Yaskawa INFORM job: DPRINT3D6.JBI

/JOB
//NAME DPRINT3D6
//POS
///NPOS 1000,0,0,0,0,0
///TOOL 9
///POSTYPE PULSE
///PULSE
C00000=29945,51705,-123586,60699,-119026,-94760,0
C00001=29937,51700,-123602,60705,-119017,-94763,0
C00002=29929,51696,-123618,60712,-119008,-94767,0
C00003=29921,51691,-123634,60719,-118999,-94770,0
C00004=29913,51687,-123649,60726,-118990,-94774,0
C00005=29905,51683,-123664,60732,-118981,-94777,0
C00006=29897,51678,-123679,60739,-118972,-94780,0
C00007=29889,51674,-123693,60746,-118964,-94782,0
C00008=29881,51670,-123708,60753,-118955,-94786,0
C00009=29873,51666,-123723,60760,-118947,-94789,0
C00010=29864,51662,-123736,60767,-118938,-94792,0
C00011=29856,51657,-123751,60774,-118930,-94795,0
C00012=29851,51655,-123762,60779,-118924,-94797,0
C00013=29843,51650,-123777,60786,-118915,-94800,0
C00014=29835,51646,-123793,60792,-118905,-94803,0
C00015=29827,51641,-123809,60799,-118896,-94807,0
C00016=29824,51639,-123816,60802,-118892,-94809,0
C00017=29807,51636,-123827,60819,-118882,-94809,0
C00018=29769,51629,-123849,60858,-118859,-94811,0
C00019=29726,51622,-123874,60903,-118835,-94812,0
C00020=29682,51615,-123900,60947,-118811,-94813,0
C00021=29646,51609,-123919,60985,-118791,-94814,0
C00022=29614,51604,-123934,61017,-118774,-94814,0
C00023=29583,51600,-123950,61050,-118758,-94814,0
C00024=29556,51596,-123961,61078,-118745,-94814,0
C00025=29529,51593,-123972,61107,-118731,-94814,0
C00026=29502,51590,-123982,61136,-118717,-94813,0
C00027=29474,51587,-123994,61164,-118704,-94813,0
C00028=29447,51583,-124005,61193,-118691,-94812,0
C00029=29424,51581,-124012,61218,-118680,-94812,0
C00030=29400,51579,-124020,61243,-118669,-94810,0
C00031=29377,51577,-124027,61267,-118658,-94810,0
C00032=29353,51574,-124035,61292,-118648,-94809,0
C00033=29333,51573,-124040,61314,-118639,-94807,0
C00034=29313,51571,-124046,61336,-118630,-94806,0
C00035=29292,51570,-124050,61358,-118622,-94805,0
C00036=29271,51568,-124055,61380,-118612,-94803,0
C00037=29251,51567,-124059,61402,-118603,-94802,0
C00038=29230,51565,-124065,61424,-118595,-94801,0
C00039=29210,51564,-124070,61446,-118586,-94800,0
C00040=29191,51563,-124073,61466,-118578,-94798,0
C00041=29173,51562,-124077,61486,-118571,-94797,0
C00042=29154,51560,-124081,61506,-118563,-94796,0
C00043=29132,51568,-124052,61533,-118568,-94785,0
C00044=29118,51573,-124034,61551,-118570,-94778,0
C00045=29103,51579,-124015,61570,-118573,-94770,0
C00046=29088,51585,-123994,61590,-118577,-94762,0
C00047=29072,51591,-123972,61610,-118580,-94754,0
C00048=29057,51597,-123951,61630,-118584,-94746,0
C00049=29042,51602,-123930,61649,-118587,-94738,0
C00050=29026,51608,-123909,61669,-118591,-94730,0
C00051=29011,51614,-123887,61689,-118594,-94722,0
C00052=28995,51621,-123864,61710,-118599,-94713,0
C00053=28978,51628,-123839,61731,-118603,-94704,0
C00054=28961,51635,-123812,61753,-118608,-94694,0
C00055=28944,51642,-123787,61775,-118612,-94684,0
C00056=28926,51650,-123758,61799,-118618,-94674,0
C00057=28907,51659,-123726,61824,-118625,-94662,0
C00058=28888,51668,-123694,61849,-118631,-94651,0
C00059=28869,51677,-123662,61874,-118638,-94639,0
C00060=28850,51686,-123631,61899,-118645,-94628,0
C00061=28831,51696,-123595,61925,-118651,-94615,0
C00062=28810,51707,-123556,61952,-118661,-94601,0
C00063=28789,51718,-123518,61980,-118669,-94588,0
C00064=28764,51733,-123464,62015,-118681,-94569,0
C00065=28738,51748,-123411,62050,-118694,-94550,0
C00066=28713,51763,-123358,62085,-118707,-94532,0
C00067=28711,51768,-123342,62089,-118712,-94527,0
C00068=28710,51773,-123323,62093,-118720,-94521,0
C00069=28708,51779,-123303,62097,-118727,-94516,0
C00070=28707,51784,-123284,62101,-118734,-94510,0
C00071=28705,51790,-123264,62105,-118742,-94504,0
C00072=28704,51796,-123245,62110,-118749,-94498,0
C00073=28703,51801,-123225,62114,-118756,-94492,0
C00074=28702,51807,-123204,62117,-118764,-94487,0
C00075=28701,51813,-123184,62121,-118772,-94481,0
C00076=28700,51819,-123163,62125,-118780,-94474,0
C00077=28699,51825,-123141,62128,-118788,-94468,0
C00078=28698,51831,-123121,62132,-118796,-94462,0
C00079=28697,51837,-123100,62136,-118804,-94456,0
C00080=28697,51843,-123078,62139,-118813,-94450,0
C00081=28696,51849,-123057,62143,-118822,-94444,0
C00082=28695,51855,-123035,62147,-118830,-94438,0
C00083=28694,51861,-123015,62150,-118838,-94431,0
C00084=28693,51867,-122994,62154,-118846,-94425,0
C00085=28693,51873,-122972,62158,-118854,-94419,0
C00086=28692,51880,-122949,62161,-118863,-94413,0
C00087=28692,51887,-122926,62164,-118872,-94406,0
C00088=28692,51893,-122903,62167,-118881,-94400,0
C00089=28692,51900,-122879,62170,-118890,-94393,0
C00090=28693,51907,-122854,62173,-118901,-94386,0
C00091=28694,51915,-122829,62176,-118911,-94379,0
C00092=28694,51922,-122805,62178,-118922,-94372,0
C00093=28695,51929,-122779,62181,-118931,-94364,0
C00094=28695,51936,-122754,62183,-118941,-94357,0
C00095=28696,51944,-122729,62186,-118951,-94350,0
C00096=28695,51949,-122708,62189,-118959,-94344,0
C00097=28697,51988,-122575,62205,-119012,-94307,0
C00098=28700,52060,-122326,62235,-119112,-94236,0
C00099=28703,52132,-122079,62265,-119211,-94166,0
C00100=22589,60303,-97251,72637,-124455,-86218,0
C00101=22532,60337,-97155,72711,-124447,-86182,0
C00102=22418,60406,-96963,72858,-124431,-86109,0
C00103=22305,60475,-96769,73005,-124414,-86036,0
C00104=22296,60482,-96752,73017,-124413,-86030,0
C00105=22287,60488,-96735,73029,-124412,-86024,0
C00106=22278,60494,-96718,73041,-124411,-86018,0
C00107=22269,60500,-96701,73053,-124411,-86011,0
C00108=22260,60506,-96684,73065,-124410,-86005,0
C00109=22251,60512,-96667,73077,-124409,-85998,0
C00110=22242,60519,-96650,73089,-124408,-85992,0
C00111=22233,60525,-96633,73101,-124408,-85986,0
C00112=22224,60531,-96615,73113,-124406,-85980,0
C00113=22215,60537,-96598,73125,-124405,-85973,0
C00114=22206,60543,-96581,73137,-124404,-85967,0
C00115=22197,60549,-96564,73149,-124404,-85961,0
C00116=22188,60555,-96547,73161,-124403,-85954,0
C00117=22180,60562,-96530,73172,-124402,-85949,0
C00118=22176,60564,-96522,73178,-124402,-85946,0
C00119=22166,60591,-96449,73200,-124414,-85924,0
C00120=22151,60635,-96326,73237,-124439,-85886,0
C00121=22136,60680,-96203,73274,-124462,-85849,0
C00122=22124,60716,-96103,73303,-124481,-85819,0
C00123=22117,60744,-96026,73324,-124496,-85795,0
C00124=22111,60768,-95959,73341,-124510,-85776,0
C00125=22106,60792,-95893,73358,-124525,-85756,0
C00126=22101,60816,-95827,73374,-124539,-85737,0
C00127=22096,60840,-95761,73391,-124552,-85717,0
C00128=22092,60858,-95711,73403,-124564,-85702,0
C00129=22090,60875,-95665,73414,-124574,-85689,0
C00130=22087,60891,-95622,73424,-124583,-85676,0
C00131=22086,60906,-95580,73433,-124594,-85665,0
C00132=22085,60921,-95539,73442,-124604,-85653,0
C00133=22083,60936,-95497,73450,-124613,-85641,0
C00134=22082,60951,-95457,73459,-124624,-85629,0
C00135=22082,60965,-95418,73466,-124634,-85618,0
C00136=22081,60979,-95379,73473,-124643,-85607,0
C00137=22081,60993,-95340,73481,-124653,-85596,0
C00138=22080,61008,-95301,73488,-124663,-85585,0
C00139=22080,61022,-95262,73496,-124673,-85574,0
C00140=22079,61036,-95223,73503,-124682,-85563,0
C00141=22079,61050,-95184,73511,-124693,-85552,0
C00142=22078,61064,-95145,73518,-124702,-85540,0
C00143=22078,61078,-95107,73525,-124712,-85530,0
C00144=22078,61092,-95070,73532,-124721,-85519,0
C00145=22077,61106,-95033,73539,-124730,-85509,0
C00146=22088,61115,-95008,73532,-124744,-85503,0
C00147=22099,61124,-94983,73526,-124757,-85498,0
C00148=22111,61133,-94958,73519,-124771,-85492,0
C00149=22123,61143,-94932,73512,-124785,-85487,0
C00150=22135,61152,-94906,73504,-124798,-85482,0
C00151=22147,61161,-94880,73497,-124813,-85477,0
C00152=22159,61171,-94854,73490,-124827,-85471,0
C00153=22171,61180,-94828,73483,-124841,-85466,0
C00154=22183,61190,-94802,73476,-124855,-85461,0
C00155=22195,61199,-94777,73468,-124870,-85455,0
C00156=22207,61209,-94751,73461,-124883,-85449,0
C00157=22219,61219,-94724,73453,-124898,-85444,0
C00158=22233,61228,-94698,73445,-124913,-85439,0
C00159=22246,61238,-94672,73436,-124928,-85434,0
C00160=22259,61248,-94645,73428,-124943,-85429,0
C00161=22277,61259,-94615,73416,-124961,-85423,0
C00162=22294,61270,-94584,73405,-124980,-85417,0
C00163=22311,61282,-94553,73393,-124999,-85411,0
C00164=22329,61293,-94522,73381,-125018,-85405,0
C00165=22346,61305,-94491,73370,-125036,-85399,0
C00166=22363,61316,-94460,73358,-125056,-85393,0
C00167=22382,61328,-94428,73345,-125075,-85387,0
C00168=22403,61340,-94395,73331,-125096,-85382,0
C00169=22428,61355,-94355,73312,-125122,-85375,0
C00170=22460,61371,-94309,73290,-125155,-85367,0
C00171=22491,61388,-94264,73267,-125186,-85359,0
C00172=22518,61402,-94226,73247,-125212,-85353,0
C00173=22552,61419,-94181,73222,-125244,-85346,0
C00174=22611,61443,-94117,73175,-125298,-85337,0
C00175=22617,61442,-94119,73169,-125300,-85339,0
C00176=22628,61441,-94122,73158,-125306,-85342,0
C00177=22639,61440,-94126,73146,-125312,-85344,0
C00178=22650,61438,-94129,73135,-125318,-85347,0
C00179=22661,61437,-94133,73123,-125325,-85350,0
C00180=22671,61436,-94136,73112,-125330,-85353,0
C00181=22682,61435,-94140,73100,-125336,-85356,0
C00182=22693,61433,-94143,73089,-125342,-85358,0
C00183=22704,61432,-94147,73077,-125348,-85361,0
C00184=22715,61431,-94150,73066,-125353,-85364,0
C00185=22726,61430,-94153,73054,-125359,-85367,0
C00186=22737,61429,-94157,73043,-125365,-85370,0
C00187=22854,61411,-94207,72918,-125423,-85404,0
C00188=22970,61393,-94257,72793,-125482,-85437,0
C00189=23087,61375,-94306,72668,-125542,-85470,0
C00190=38516,60450,-97093,77282,-121914,-85527,0
C00191=38540,60506,-96937,77284,-121963,-85486,0
C00192=38587,60619,-96625,77287,-122064,-85402,0
C00193=38635,60733,-96312,77291,-122166,-85319,0
C00194=38639,60742,-96286,77291,-122174,-85312,0
C00195=38643,60752,-96261,77291,-122183,-85306,0
C00196=38648,60761,-96236,77290,-122191,-85299,0
C00197=38652,60770,-96210,77290,-122200,-85292,0
C00198=38657,60779,-96185,77290,-122208,-85285,0
C00199=38661,60789,-96159,77290,-122217,-85279,0
C00200=38665,60798,-96134,77290,-122225,-85272,0
C00201=38670,60807,-96108,77289,-122235,-85266,0
C00202=38674,60816,-96083,77289,-122243,-85259,0
C00203=38679,60826,-96057,77289,-122251,-85252,0
C00204=38683,60835,-96032,77289,-122260,-85245,0
C00205=38687,60844,-96006,77289,-122268,-85238,0
C00206=38692,60854,-95981,77288,-122277,-85232,0
C00207=38696,60862,-95956,77288,-122285,-85226,0
C00208=38698,60867,-95944,77288,-122290,-85222,0
C00209=38725,60883,-95901,77269,-122316,-85213,0
C00210=38769,60909,-95831,77237,-122360,-85199,0
C00211=38814,60934,-95761,77204,-122403,-85186,0
C00212=38851,60954,-95706,77178,-122439,-85176,0
C00213=38879,60969,-95667,77156,-122466,-85168,0
C00214=38904,60981,-95636,77137,-122488,-85163,0
C00215=38929,60992,-95605,77118,-122510,-85158,0
C00216=38954,61003,-95574,77099,-122533,-85152,0
C00217=38978,61015,-95543,77080,-122555,-85147,0
C00218=38997,61023,-95521,77065,-122572,-85143,0
C00219=39015,61030,-95501,77051,-122587,-85140,0
C00220=39031,61037,-95483,77038,-122602,-85137,0
C00221=39047,61042,-95468,77025,-122616,-85135,0
C00222=39063,61048,-95453,77012,-122629,-85133,0
C00223=39079,61054,-95438,76999,-122642,-85131,0
C00224=39094,61059,-95424,76986,-122655,-85129,0
C00225=39110,61063,-95412,76974,-122668,-85128,0
C00226=39125,61068,-95399,76961,-122680,-85126,0
C00227=39140,61073,-95387,76948,-122692,-85125,0
C00228=39155,61077,-95375,76935,-122705,-85124,0
C00229=39170,61082,-95362,76923,-122717,-85122,0
C00230=39185,61087,-95349,76910,-122730,-85121,0
C00231=39200,61091,-95337,76897,-122741,-85119,0
C00232=39216,61096,-95325,76884,-122754,-85118,0
C00233=39230,61100,-95313,76872,-122767,-85117,0
C00234=39245,61104,-95302,76860,-122778,-85116,0
C00235=39259,61109,-95291,76847,-122790,-85115,0
C00236=39272,61102,-95309,76832,-122793,-85122,0
C00237=39285,61095,-95327,76816,-122796,-85129,0
C00238=39298,61088,-95347,76800,-122800,-85137,0
C00239=39312,61081,-95368,76783,-122805,-85144,0
C00240=39325,61074,-95388,76767,-122808,-85152,0
C00241=39339,61066,-95409,76750,-122811,-85161,0
C00242=39353,61059,-95429,76734,-122815,-85168,0
C00243=39366,61051,-95450,76717,-122818,-85176,0
C00244=39380,61044,-95470,76700,-122823,-85184,0
C00245=39393,61037,-95491,76684,-122826,-85192,0
C00246=39407,61029,-95511,76667,-122830,-85199,0
C00247=39421,61021,-95534,76650,-122833,-85208,0
C00248=39435,61013,-95557,76632,-122837,-85217,0
C00249=39449,61004,-95581,76614,-122840,-85226,0
C00250=39463,60996,-95604,76597,-122842,-85235,0
C00251=39481,60984,-95636,76575,-122846,-85246,0
C00252=39498,60973,-95668,76553,-122849,-85257,0
C00253=39515,60962,-95699,76531,-122853,-85269,0
C00254=39532,60950,-95731,76509,-122855,-85281,0
C00255=39549,60939,-95763,76487,-122859,-85292,0
C00256=39566,60927,-95794,76465,-122862,-85304,0
C00257=39584,60915,-95829,76441,-122864,-85317,0
C00258=39603,60901,-95868,76416,-122868,-85331,0
C00259=39626,60883,-95917,76386,-122870,-85348,0
C00260=39653,60861,-95978,76349,-122872,-85369,0
C00261=39680,60840,-96038,76313,-122875,-85391,0
C00262=39702,60821,-96089,76282,-122876,-85408,0
C00263=39730,60797,-96156,76244,-122877,-85432,0
C00264=39772,60754,-96276,76183,-122875,-85472,0
C00265=39773,60749,-96290,76180,-122872,-85476,0
C00266=39775,60739,-96316,76173,-122867,-85484,0
C00267=39777,60730,-96343,76167,-122862,-85492,0
C00268=39779,60720,-96369,76161,-122856,-85500,0
C00269=39781,60711,-96396,76155,-122852,-85508,0
C00270=39782,60701,-96422,76149,-122846,-85516,0
C00271=39784,60692,-96449,76143,-122841,-85524,0
C00272=39786,60682,-96475,76136,-122836,-85531,0
C00273=39788,60672,-96501,76130,-122831,-85539,0
C00274=39790,60663,-96528,76124,-122825,-85547,0
C00275=39792,60653,-96554,76118,-122821,-85555,0
C00276=39793,60644,-96581,76112,-122815,-85563,0
C00277=39808,60540,-96867,76051,-122755,-85647,0
C00278=39822,60438,-97152,75990,-122695,-85730,0
C00279=39836,60335,-97436,75930,-122636,-85814,0
C00280=30587,54971,-112893,83159,-114119,-89355,0
C00281=30599,54742,-113602,83076,-113987,-89576,0
C00282=26102,60146,-97730,68982,-126367,-86955,0
C00283=25840,59681,-99025,69012,-125831,-87267,0
C00284=25634,59454,-99658,69109,-125527,-87407,0
C00285=25332,58798,-101506,69089,-124805,-87871,0
C00286=25979,60253,-97431,69165,-126385,-86850,0
C00287=30587,54971,-112892,83159,-114119,-89355,0
C00288=31709,55377,-111663,82144,-114929,-89073,0
C00289=25839,57975,-103866,68149,-124352,-88615,0
C00290=26365,57183,-106175,67203,-123890,-89348,0
C00291=32807,55804,-110382,81171,-115756,-88784,0
C00292=33879,56254,-109050,80240,-116598,-88487,0
C00293=26912,56421,-108432,66247,-123417,-90067,0
C00294=27480,55689,-110642,65280,-122933,-90775,0
C00295=34926,56725,-107667,79351,-117457,-88183,0
C00296=35949,57218,-106233,78506,-118333,-87871,0
C00297=28070,54985,-112806,64301,-122438,-91471,0
C00298=28684,54309,-114927,63309,-121930,-92157,0
C00299=36947,57735,-104747,77703,-119224,-87551,0
C00300=37852,58236,-103319,76997,-120066,-87245,0
C00301=37910,58216,-103377,76930,-120084,-87270,0
C00302=29401,53804,-116547,62283,-121613,-92717,0
C00303=29691,53808,-116540,61968,-121730,-92760,0
C00304=30366,53748,-116745,61199,-121915,-92922,0
C00305=38739,58035,-103915,76018,-120418,-87536,0
C00306=38801,58025,-103945,75951,-120444,-87552,0
C00307=39443,58021,-103971,75297,-120792,-87646,0
C00308=39602,58044,-103908,75146,-120896,-87649,0
C00309=31268,53565,-117352,60117,-122023,-93230,0
C00310=31586,53466,-117679,59719,-122012,-93369,0
C00311=32325,53708,-116909,59020,-122601,-93280,0
C00312=40396,57540,-105383,74115,-120944,-88187,0
C00313=41188,56884,-107325,73008,-120835,-88860,0
C00314=33470,54107,-115653,57950,-123551,-93138,0
C00315=34587,54528,-114347,56920,-124521,-92992,0
C00316=42006,56254,-109216,71875,-120713,-89524,0
C00317=42851,55650,-111059,70716,-120580,-90176,0
C00318=35677,54970,-112991,55932,-125513,-92844,0
C00319=43402,51305,-125329,68233,-116168,-94477,0
C00320=43725,55072,-112853,69529,-120434,-90818,0
C00321=44627,54518,-114601,68312,-120275,-91449,0
C00322=44483,51740,-123805,67237,-117079,-94137,0
C00323=45527,52199,-122237,66296,-118013,-93796,0
C00324=45537,52695,-120546,66506,-118620,-93300,0
C00325=45537,52633,-120569,66515,-118645,-93280,0
C00326=46697,53753,-116919,65763,-120389,-92380,0
C00327=46484,53451,-117891,65855,-119960,-92629,0
C00328=46391,53159,-118843,65822,-119586,-92891,0
C00329=46413,52869,-119803,65666,-119250,-93171,0
C00330=46552,52597,-120719,65391,-118971,-93455,0
C00331=46800,52351,-121557,65008,-118755,-93730,0
C00332=31582,53062,-118822,59567,-121584,-93654,0
C00333=31079,53242,-118223,60209,-121640,-93412,0
C00334=30561,53361,-117825,60837,-121604,-93223,0
C00335=30009,53428,-117599,61476,-121481,-93076,0
C00336=29447,53437,-117559,62097,-121280,-92979,0
C00337=28896,53391,-117698,62679,-121012,-92936,0
C00338=24566,59142,-100391,70091,-124739,-87405,0
C00339=24937,59442,-99553,69860,-125191,-87233,0
C00340=25205,59777,-98620,69755,-125616,-87019,0
C00341=25384,60157,-97564,69765,-126028,-86756,0
C00342=25469,60567,-96432,69890,-126406,-86456,0
C00343=29650,54961,-112750,84133,-113691,-89204,0
C00344=37685,58554,-102273,77329,-120238,-86893,0
C00345=38136,58340,-102891,76787,-120350,-87132,0
C00346=38606,58212,-103267,76260,-120523,-87303,0
C00347=39106,58161,-103425,75733,-120765,-87417,0
C00348=39613,58188,-103358,75231,-121064,-87466,0
C00349=40132,58300,-103047,74754,-121431,-87448,0
C00350=46626,53790,-116798,65857,-120402,-92336,0
C00351=48080,52338,-121638,63597,-119184,-93923,0
C00352=31354,52451,-120852,59527,-120671,-94173,0
C00353=31201,52571,-120444,59753,-120784,-94039,0
C00354=30927,52714,-119961,60125,-120883,-93865,0
C00355=30607,52827,-119581,60531,-120921,-93713,0
C00356=30254,52906,-119311,60958,-120900,-93585,0
C00357=29878,52950,-119159,61393,-120821,-93487,0
C00358=29495,52956,-119132,61816,-120689,-93424,0
C00359=29122,52926,-119226,62211,-120513,-93395,0
C00360=29011,52905,-119293,62324,-120446,-93397,0
C00361=28935,52897,-119318,62403,-120407,-93394,0
C00362=28456,52795,-119645,62881,-120103,-93418,0
C00363=23544,59431,-99566,71281,-124398,-87003,0
C00364=23825,59520,-99321,71038,-124627,-86981,0
C00365=24097,59665,-98918,70832,-124897,-86913,0
C00366=24327,59854,-98395,70691,-125179,-86805,0
C00367=24510,60081,-97764,70620,-125464,-86660,0
C00368=24634,60340,-97049,70624,-125739,-86481,0
C00369=24696,60619,-96279,70704,-125995,-86277,0
C00370=24693,60909,-95482,70856,-126218,-86054,0
C00371=24624,61196,-94694,71073,-126396,-85821,0
C00372=28555,55200,-111997,85310,-113265,-88883,0
C00373=37805,59412,-99847,77570,-120870,-86202,0
C00374=37976,59213,-100409,77316,-120843,-86388,0
C00375=38214,59036,-100913,77004,-120864,-86567,0
C00376=38493,58902,-101297,76668,-120935,-86716,0
C00377=38807,58815,-101551,76316,-121054,-86832,0
C00378=39141,58780,-101658,75966,-121220,-86908,0
C00379=39481,58798,-101612,75632,-121426,-86942,0
C00380=39812,58871,-101412,75331,-121665,-86931,0
C00381=40119,58996,-101065,75077,-121928,-86874,0
C00382=40308,59117,-100727,74941,-122122,-86804,0
C00383=47910,53822,-116729,64476,-120945,-92502,0
C00384=47717,53706,-117098,64631,-120735,-92578,0
C00385=47517,53528,-117667,64766,-120449,-92711,0
C00386=47387,53338,-118283,64818,-120175,-92868,0
C00387=47331,53142,-118926,64789,-119919,-93044,0
C00388=47352,52947,-119570,64677,-119690,-93231,0
C00389=47450,52764,-120182,64485,-119502,-93420,0
C00390=47620,52599,-120739,64223,-119357,-93603,0
C00391=47693,52555,-120892,64122,-119327,-93657,0
C00392=47732,52522,-121003,64065,-119300,-93693,0
C00393=48011,52374,-121513,63690,-119207,-93878,0
C00394=48242,52920,-119683,63689,-119983,-93387,0
C00395=48338,52828,-119993,63541,-119902,-93488,0
C00396=48398,52792,-120115,63459,-119878,-93531,0
C00397=48426,52769,-120192,63417,-119859,-93557,0
C00398=48563,52696,-120443,63232,-119814,-93647,0
C00399=48728,52637,-120643,63024,-119797,-93727,0
C00400=48914,52596,-120787,62799,-119810,-93794,0
C00401=49115,52574,-120866,62568,-119851,-93844,0
C00402=49652,52569,-120900,61974,-120029,-93930,0
C00403=30732,51817,-123013,59918,-119564,-94680,0
C00404=30754,52010,-122343,59984,-119849,-94498,0
C00405=30718,52122,-121960,60075,-119995,-94386,0
C00406=30636,52229,-121591,60217,-120118,-94272,0
C00407=30516,52322,-121274,60393,-120205,-94167,0
C00408=30359,52403,-120996,60605,-120263,-94068,0
C00409=30175,52467,-120777,60838,-120286,-93980,0
C00410=29972,52511,-120623,61082,-120275,-93908,0
C00411=29757,52536,-120536,61330,-120233,-93853,0
C00412=29540,52539,-120521,61571,-120160,-93818,0
C00413=29329,52522,-120574,61795,-120064,-93802,0
C00414=29239,52506,-120627,61887,-120010,-93804,0
C00415=29184,52500,-120645,61944,-119983,-93802,0
C00416=28994,52461,-120775,62135,-119863,-93812,0
C00417=28822,52404,-120962,62298,-119728,-93840,0
C00418=28675,52334,-121198,62426,-119583,-93887,0
C00419=28559,52252,-121475,62516,-119434,-93949,0
C00420=28349,52018,-122269,62640,-119049,-94147,0
C00421=22462,60078,-97747,72692,-124270,-86314,0
C00422=22881,59971,-98051,72218,-124434,-86468,0
C00423=23049,59957,-98090,72041,-124521,-86506,0
C00424=23127,59964,-98072,71965,-124572,-86514,0
C00425=23172,59963,-98076,71919,-124597,-86522,0
C00426=23344,59987,-98011,71757,-124716,-86532,0
C00427=23510,60040,-97866,71615,-124852,-86519,0
C00428=23662,60123,-97638,71502,-125005,-86481,0
C00429=23793,60231,-97341,71423,-125164,-86419,0
C00430=23898,60361,-96980,71383,-125327,-86336,0
C00431=23971,60511,-96568,71384,-125484,-86232,0
C00432=24009,60673,-96122,71427,-125630,-86114,0
C00433=24009,60842,-95658,71512,-125759,-85984,0
C00434=23971,61010,-95195,71636,-125862,-85848,0
C00435=23919,61122,-94888,71746,-125915,-85752,0
C00436=23874,61195,-94688,71828,-125943,-85689,0
C00437=23749,61329,-94321,72021,-125966,-85564,0
C00438=23379,61600,-93579,72527,-125937,-85292,0
C00439=38290,60454,-96953,77539,-121827,-85431,0
C00440=38275,60082,-97984,77393,-121581,-85727,0
C00441=38302,59941,-98375,77305,-121507,-85843,0
C00442=38330,59880,-98546,77251,-121484,-85896,0
C00443=38339,59843,-98649,77226,-121467,-85928,0
C00444=38410,59712,-99017,77099,-121423,-86044,0
C00445=38513,59593,-99352,76946,-121407,-86155,0
C00446=38647,59493,-99635,76769,-121419,-86255,0
C00447=38804,59416,-99855,76579,-121460,-86340,0
C00448=38982,59366,-100000,76381,-121530,-86406,0
C00449=39172,59345,-100061,76182,-121627,-86450,0
C00450=39366,59356,-100035,75993,-121746,-86470,0
C00451=39557,59399,-99918,75821,-121886,-86463,0
C00452=39736,59473,-99714,75675,-122041,-86430,0
C00453=39847,59544,-99515,75597,-122155,-86389,0
C00454=39915,59600,-99361,75553,-122233,-86354,0
C00455=40028,59737,-98979,75503,-122394,-86261,0
C00456=40217,60115,-97929,75486,-122764,-85987,0
C00457=49320,53737,-117041,62893,-121389,-92800,0
C00458=48930,53677,-117223,63292,-121168,-92792,0
C00459=48720,53621,-117399,63495,-121020,-92810,0
C00460=48536,53546,-117638,63661,-120859,-92850,0
C00461=48384,53455,-117930,63784,-120692,-92910,0
C00462=48270,53353,-118260,63860,-120526,-92987,0
C00463=48199,53245,-118611,63888,-120367,-93077,0
C00464=48169,53132,-118979,63868,-120219,-93176,0
C00465=48184,53023,-119341,63801,-120090,-93281,0
C00466=48214,52969,-119521,63742,-120034,-93336,0
C00467=48109,52838,-119955,63796,-119832,-93446,0
C00468=49394,53547,-117657,62721,-121185,-92983,0
C00469=49490,53541,-117679,62612,-121214,-93003,0
C00470=49683,53530,-117722,62395,-121272,-93044,0
C00471=49785,53524,-117745,62280,-121303,-93066,0
C00472=49799,53522,-117748,62265,-121306,-93069,0
C00473=49813,53521,-117753,62249,-121309,-93072,0
C00474=49827,53520,-117756,62233,-121313,-93075,0
C00475=49840,53519,-117761,62217,-121318,-93079,0
C00476=49852,53518,-117764,62204,-121320,-93082,0
C00477=49863,53517,-117769,62191,-121322,-93085,0
C00478=49876,53515,-117774,62176,-121326,-93088,0
C00479=49889,53514,-117779,62161,-121329,-93091,0
C00480=49903,53512,-117784,62146,-121331,-93095,0
C00481=49916,53511,-117790,62130,-121335,-93098,0
C00482=49929,53509,-117794,62115,-121338,-93101,0
C00483=49943,53508,-117800,62099,-121342,-93105,0
C00484=49956,53506,-117805,62084,-121344,-93108,0
C00485=49969,53505,-117810,62069,-121347,-93112,0
C00486=49983,53503,-117815,62053,-121351,-93115,0
C00487=49993,53502,-117819,62042,-121353,-93118,0
C00488=50003,53501,-117824,62030,-121354,-93121,0
C00489=50045,53479,-117898,61973,-121343,-93148,0
C00490=50081,53458,-117964,61923,-121330,-93172,0
C00491=50118,53438,-118031,61873,-121319,-93196,0
C00492=50148,53421,-118090,61831,-121307,-93216,0
C00493=50173,53406,-118138,61797,-121298,-93234,0
C00494=50192,53393,-118181,61770,-121289,-93249,0
C00495=50212,53380,-118224,61742,-121280,-93264,0
C00496=50231,53367,-118268,61714,-121269,-93278,0
C00497=50251,53354,-118311,61686,-121260,-93294,0
C00498=50271,53341,-118354,61658,-121251,-93309,0
C00499=50283,53331,-118386,61639,-121243,-93319,0
C00500=50296,53322,-118417,61621,-121236,-93330,0
C00501=50309,53312,-118449,61602,-121228,-93341,0
C00502=50321,53303,-118480,61585,-121221,-93351,0
C00503=50332,53293,-118511,61568,-121213,-93361,0
C00504=50343,53284,-118541,61551,-121205,-93371,0
C00505=50355,53275,-118572,61534,-121197,-93382,0
C00506=50366,53265,-118603,61517,-121189,-93392,0
C00507=50377,53256,-118634,61500,-121181,-93402,0
C00508=50389,53247,-118665,61483,-121174,-93412,0
C00509=50399,53238,-118694,61467,-121166,-93422,0
C00510=50408,53229,-118723,61453,-121159,-93431,0
C00511=50417,53221,-118750,61439,-121151,-93440,0
C00512=50427,53213,-118778,61425,-121143,-93450,0
C00513=50436,53204,-118805,61411,-121136,-93458,0
C00514=50443,53197,-118831,61399,-121129,-93466,0
C00515=50450,53189,-118856,61387,-121121,-93475,0
C00516=50458,53182,-118881,61375,-121114,-93483,0
C00517=50465,53174,-118905,61364,-121107,-93491,0
C00518=50473,53166,-118931,61352,-121100,-93499,0
C00519=50480,53159,-118956,61340,-121093,-93507,0
C00520=50487,53151,-118981,61328,-121087,-93515,0
C00521=50495,53144,-119007,61317,-121078,-93523,0
C00522=50502,53136,-119031,61305,-121072,-93531,0
C00523=50497,53130,-119054,61307,-121061,-93537,0
C00524=50490,53120,-119084,61310,-121046,-93544,0
C00525=50483,53111,-119115,61314,-121033,-93551,0
C00526=50476,53102,-119144,61317,-121018,-93558,0
C00527=50469,53093,-119174,61321,-121003,-93566,0
C00528=50461,53084,-119204,61325,-120989,-93573,0
C00529=50451,53073,-119240,61330,-120970,-93581,0
C00530=50441,53062,-119277,61336,-120953,-93590,0
C00531=50431,53051,-119312,61342,-120935,-93598,0
C00532=50421,53040,-119348,61348,-120918,-93607,0
C00533=50412,53029,-119385,61353,-120899,-93616,0
C00534=50401,53018,-119420,61359,-120882,-93624,0
C00535=50390,53006,-119457,61366,-120862,-93632,0
C00536=50378,52995,-119496,61374,-120843,-93642,0
C00537=50366,52983,-119535,61382,-120823,-93650,0
C00538=50351,52970,-119579,61392,-120800,-93660,0
C00539=50335,52955,-119625,61403,-120776,-93671,0
C00540=50318,52941,-119672,61415,-120752,-93682,0
C00541=50301,52927,-119718,61427,-120728,-93692,0
C00542=50292,52924,-119729,61436,-120720,-93693,0
C00543=50282,52921,-119740,61444,-120712,-93695,0
C00544=50273,52917,-119750,61454,-120704,-93697,0
C00545=50263,52914,-119762,61463,-120697,-93698,0
C00546=50252,52911,-119772,61473,-120689,-93700,0
C00547=50241,52907,-119782,61483,-120680,-93701,0
C00548=50230,52904,-119794,61494,-120672,-93703,0
C00549=50220,52901,-119804,61504,-120664,-93704,0
C00550=50209,52897,-119816,61514,-120656,-93706,0
C00551=50198,52894,-119826,61525,-120648,-93707,0
C00552=50186,52891,-119836,61536,-120639,-93708,0
C00553=50175,52888,-119847,61548,-120631,-93709,0
C00554=50163,52884,-119857,61559,-120623,-93710,0
C00555=50152,52881,-119867,61570,-120614,-93711,0
C00556=50140,52878,-119878,61581,-120606,-93712,0
C00557=50128,52875,-119888,61592,-120598,-93714,0
C00558=50117,52872,-119897,61604,-120590,-93715,0
C00559=50105,52869,-119907,61615,-120582,-93716,0
C00560=50094,52865,-119918,61626,-120574,-93717,0
C00561=50082,52862,-119928,61638,-120565,-93718,0
C00562=50071,52859,-119939,61649,-120557,-93719,0
C00563=50059,52856,-119949,61660,-120549,-93721,0
C00564=50047,52853,-119959,61672,-120541,-93722,0
C00565=50034,52850,-119968,61684,-120533,-93723,0
C00566=50022,52847,-119978,61697,-120525,-93724,0
C00567=50008,52844,-119988,61710,-120515,-93725,0
C00568=49994,52841,-119998,61725,-120506,-93725,0
C00569=49979,52837,-120007,61740,-120497,-93726,0
C00570=49964,52834,-120018,61755,-120488,-93726,0
C00571=49949,52831,-120028,61770,-120479,-93727,0
C00572=49934,52828,-120037,61784,-120468,-93728,0
C00573=49919,52825,-120048,61799,-120459,-93728,0
C00574=49905,52822,-120058,61814,-120450,-93729,0
C00575=49890,52819,-120068,61829,-120441,-93730,0
C00576=49875,52816,-120078,61844,-120432,-93730,0
C00577=49858,52812,-120088,61861,-120421,-93730,0
C00578=49803,52804,-120115,61918,-120390,-93730,0
C00579=49709,52789,-120161,62014,-120340,-93730,0
C00580=30345,51835,-122941,60354,-119464,-94607,0
C00581=30254,51752,-123229,60417,-119316,-94675,0
C00582=30162,51670,-123514,60480,-119167,-94742,0
C00583=30155,51664,-123533,60486,-119156,-94747,0
C00584=30148,51658,-123553,60491,-119146,-94752,0
C00585=30141,51653,-123573,60496,-119135,-94756,0
C00586=30134,51647,-123593,60502,-119125,-94761,0
C00587=30127,51642,-123610,60507,-119116,-94765,0
C00588=30121,51637,-123626,60511,-119107,-94769,0
C00589=30114,51632,-123645,60517,-119097,-94773,0
C00590=30106,51627,-123663,60523,-119087,-94777,0
C00591=30098,51622,-123681,60529,-119077,-94781,0
C00592=30090,51616,-123701,60535,-119066,-94785,0
C00593=30083,51611,-123719,60541,-119056,-94789,0
C00594=30075,51605,-123739,60547,-119046,-94794,0
C00595=30067,51600,-123757,60553,-119035,-94798,0
C00596=30059,51594,-123776,60560,-119025,-94802,0
C00597=30051,51589,-123795,60566,-119015,-94807,0
C00598=30044,51584,-123811,60571,-119005,-94810,0
C00599=30038,51580,-123826,60576,-118997,-94814,0
C00600=30035,51578,-123833,60579,-118993,-94815,0
C00601=30003,51571,-123856,60611,-118973,-94817,0
C00602=29951,51561,-123890,60665,-118942,-94820,0
C00603=29898,51551,-123925,60718,-118910,-94823,0
C00604=29845,51541,-123959,60772,-118879,-94825,0
C00605=29807,51535,-123981,60811,-118857,-94827,0
C00606=29772,51529,-124000,60847,-118838,-94827,0
C00607=29739,51525,-124016,60882,-118820,-94827,0
C00608=29706,51520,-124032,60916,-118803,-94827,0
C00609=29674,51515,-124047,60950,-118787,-94827,0
C00610=29641,51511,-124063,60984,-118770,-94827,0
C00611=29613,51507,-124075,61013,-118755,-94827,0
C00612=29589,51505,-124084,61038,-118743,-94827,0
C00613=29566,51502,-124093,61063,-118732,-94826,0
C00614=29543,51499,-124101,61087,-118722,-94825,0
C00615=29520,51497,-124108,61111,-118711,-94824,0
C00616=29498,51495,-124115,61135,-118701,-94824,0
C00617=29475,51493,-124121,61159,-118691,-94823,0
C00618=29453,51491,-124128,61183,-118680,-94821,0
C00619=29430,51489,-124136,61206,-118670,-94821,0
C00620=29408,51487,-124142,61230,-118660,-94820,0
C00621=29385,51485,-124149,61254,-118650,-94818,0
C00622=29365,51484,-124154,61276,-118641,-94817,0
C00623=29345,51482,-124158,61297,-118633,-94816,0
C00624=29326,51481,-124163,61319,-118625,-94814,0
C00625=29306,51479,-124167,61340,-118616,-94813,0
C00626=29287,51478,-124171,61360,-118609,-94812,0
C00627=29269,51478,-124173,61379,-118602,-94810,0
C00628=29252,51477,-124177,61398,-118595,-94809,0
C00629=29234,51476,-124179,61417,-118588,-94807,0
C00630=29216,51475,-124181,61436,-118581,-94806,0
C00631=29199,51474,-124183,61456,-118574,-94804,0
C00632=29181,51473,-124186,61475,-118568,-94802,0
C00633=29164,51473,-124189,61494,-118561,-94800,0
C00634=29146,51472,-124192,61513,-118554,-94799,0
C00635=29137,51471,-124193,61522,-118550,-94798,0
C00636=29125,51475,-124178,61537,-118553,-94793,0
C00637=29110,51481,-124157,61556,-118556,-94785,0
C00638=29095,51487,-124135,61576,-118560,-94777,0
C00639=29080,51493,-124115,61595,-118563,-94769,0
C00640=29065,51499,-124093,61615,-118568,-94760,0
C00641=29050,51505,-124072,61634,-118571,-94752,0
C00642=29032,51513,-124044,61657,-118576,-94742,0
C00643=29015,51520,-124017,61680,-118581,-94733,0
C00644=28997,51528,-123989,61703,-118586,-94722,0
C00645=28980,51536,-123962,61725,-118592,-94712,0
C00646=28962,51543,-123935,61748,-118596,-94702,0
C00647=28945,51551,-123908,61771,-118602,-94692,0
C00648=28927,51559,-123878,61795,-118608,-94681,0
C00649=28908,51568,-123846,61819,-118615,-94670,0
C00650=28890,51577,-123813,61844,-118622,-94658,0
C00651=28870,51588,-123777,61870,-118630,-94645,0
C00652=28849,51599,-123736,61899,-118639,-94630,0
C00653=28827,51611,-123695,61928,-118648,-94616,0
C00654=28806,51622,-123654,61957,-118657,-94601,0
C00655=28803,51628,-123635,61962,-118664,-94596,0
C00656=28800,51633,-123618,61967,-118670,-94590,0
C00657=28798,51638,-123600,61973,-118677,-94585,0
C00658=28795,51643,-123581,61978,-118684,-94579,0
C00659=28793,51649,-123561,61983,-118691,-94574,0
C00660=28790,51654,-123541,61988,-118697,-94567,0
C00661=28788,51660,-123522,61993,-118704,-94561,0
C00662=28786,51666,-123502,61999,-118711,-94556,0
C00663=28783,51671,-123481,62004,-118719,-94550,0
C00664=28781,51677,-123462,62009,-118726,-94543,0
C00665=28780,51683,-123440,62013,-118734,-94537,0
C00666=28778,51689,-123419,62018,-118742,-94531,0
C00667=28776,51695,-123399,62023,-118749,-94525,0
C00668=28774,51701,-123378,62027,-118757,-94518,0
C00669=28772,51707,-123357,62032,-118765,-94513,0
C00670=28771,51713,-123335,62037,-118773,-94506,0
C00671=28769,51719,-123315,62041,-118780,-94500,0
C00672=28767,51725,-123294,62046,-118788,-94494,0
C00673=28765,51731,-123273,62051,-118796,-94488,0
C00674=28764,51737,-123253,62055,-118804,-94481,0
C00675=28762,51743,-123231,62060,-118811,-94475,0
C00676=28760,51749,-123210,62065,-118819,-94469,0
C00677=28759,51755,-123188,62069,-118827,-94463,0
C00678=28758,51761,-123166,62073,-118835,-94456,0
C00679=28756,51768,-123145,62077,-118845,-94450,0
C00680=28756,51774,-123122,62081,-118854,-94443,0
C00681=28755,51782,-123095,62085,-118863,-94435,0
C00682=28755,51789,-123070,62089,-118873,-94429,0
C00683=28754,51797,-123044,62093,-118884,-94421,0
C00684=28754,51804,-123018,62097,-118894,-94413,0
C00685=28753,51811,-122993,62101,-118904,-94406,0
C00686=28753,51819,-122967,62105,-118913,-94399,0
C00687=28752,51826,-122941,62108,-118924,-94391,0
C00688=28752,51834,-122915,62112,-118934,-94384,0
C00689=28752,51841,-122890,62116,-118944,-94376,0
C00690=28752,51849,-122861,62120,-118956,-94368,0
C00691=28756,51876,-122768,62128,-118994,-94343,0
C00692=28763,51921,-122611,62141,-119058,-94299,0
C00693=22641,60308,-97114,72623,-124545,-86164,0
C00694=22587,60350,-96995,72699,-124544,-86121,0
C00695=22478,60436,-96756,72849,-124543,-86037,0
C00696=22420,60483,-96627,72930,-124543,-85990,0
C00697=22412,60490,-96607,72942,-124543,-85984,0
C00698=22404,60497,-96587,72953,-124544,-85977,0
C00699=22396,60504,-96567,72965,-124544,-85970,0
C00700=22388,60511,-96548,72976,-124544,-85963,0
C00701=22380,60518,-96528,72988,-124545,-85956,0
C00702=22372,60526,-96508,73000,-124545,-85949,0
C00703=22364,60533,-96489,73011,-124545,-85942,0
C00704=22355,60540,-96469,73023,-124547,-85935,0
C00705=22347,60547,-96449,73034,-124547,-85929,0
C00706=22339,60554,-96429,73046,-124547,-85922,0
C00707=22333,60561,-96411,73055,-124548,-85915,0
C00708=22326,60567,-96393,73065,-124549,-85910,0
C00709=22319,60574,-96375,73075,-124549,-85903,0
C00710=22313,60580,-96357,73085,-124550,-85897,0
C00711=22306,60587,-96339,73094,-124551,-85891,0
C00712=22300,60593,-96320,73104,-124552,-85885,0
C00713=22294,60600,-96302,73113,-124554,-85878,0
C00714=22287,60607,-96282,73124,-124554,-85871,0
C00715=22279,60614,-96262,73135,-124555,-85865,0
C00716=22271,60622,-96242,73146,-124555,-85858,0
C00717=22264,60629,-96223,73157,-124556,-85851,0
C00718=22256,60636,-96203,73168,-124556,-85845,0
C00719=22249,60643,-96184,73179,-124557,-85838,0
C00720=22243,60649,-96167,73188,-124558,-85832,0
C00721=22237,60656,-96148,73197,-124559,-85826,0
C00722=22231,60662,-96130,73207,-124560,-85820,0
C00723=22225,60669,-96112,73216,-124562,-85813,0
C00724=22218,60675,-96094,73225,-124562,-85808,0
C00725=22212,60682,-96076,73235,-124563,-85801,0
C00726=22206,60688,-96058,73244,-124564,-85795,0
C00727=22201,60695,-96040,73253,-124565,-85790,0
C00728=22195,60701,-96022,73261,-124567,-85783,0
C00729=22190,60708,-96004,73270,-124568,-85777,0
C00730=22184,60714,-95986,73279,-124570,-85771,0
C00731=22178,60721,-95968,73288,-124571,-85765,0
C00732=22176,60724,-95959,73292,-124572,-85762,0
C00733=22172,60738,-95922,73302,-124579,-85751,0
C00734=22166,60765,-95848,73321,-124595,-85729,0
C00735=22161,60788,-95783,73337,-124609,-85710,0
C00736=22158,60808,-95729,73350,-124621,-85694,0
C00737=22154,60828,-95674,73363,-124633,-85678,0
C00738=22152,60846,-95623,73375,-124644,-85664,0
C00739=22150,60864,-95575,73386,-124656,-85650,0
C00740=22148,60881,-95527,73396,-124667,-85636,0
C00741=22146,60898,-95480,73407,-124679,-85622,0
C00742=22144,60916,-95432,73417,-124689,-85608,0
C00743=22142,60933,-95384,73428,-124701,-85595,0
C00744=22140,60949,-95340,73437,-124711,-85582,0
C00745=22139,60964,-95299,73445,-124721,-85570,0
C00746=22138,60979,-95259,73453,-124732,-85559,0
C00747=22138,60994,-95218,73461,-124741,-85547,0
C00748=22137,61009,-95177,73469,-124751,-85535,0
C00749=22136,61021,-95144,73476,-124760,-85526,0
C00750=22136,61031,-95117,73480,-124767,-85518,0
C00751=22141,61035,-95105,73478,-124773,-85516,0
C00752=22151,61044,-95081,73472,-124785,-85510,0
C00753=22161,61053,-95057,73467,-124797,-85505,0
C00754=22170,61061,-95033,73461,-124810,-85500,0
C00755=22180,61070,-95009,73456,-124821,-85495,0
C00756=22190,61079,-94986,73451,-124834,-85490,0
C00757=22200,61088,-94962,73446,-124845,-85484,0
C00758=22209,61096,-94938,73440,-124858,-85479,0
C00759=22220,61105,-94913,73434,-124871,-85474,0
C00760=22231,61114,-94889,73428,-124884,-85469,0
C00761=22242,61124,-94864,73421,-124897,-85463,0
C00762=22253,61133,-94839,73415,-124910,-85459,0
C00763=22264,61142,-94814,73408,-124924,-85454,0
C00764=22276,61151,-94788,73401,-124938,-85448,0
C00765=22290,61162,-94760,73392,-124953,-85443,0
C00766=22304,61172,-94732,73383,-124970,-85437,0
C00767=22317,61182,-94705,73375,-124986,-85431,0
C00768=22331,61192,-94676,73366,-125001,-85425,0
C00769=22345,61203,-94648,73358,-125017,-85420,0
C00770=22358,61213,-94620,73349,-125033,-85414,0
C00771=22373,61224,-94591,73340,-125049,-85408,0
C00772=22389,61235,-94562,73329,-125066,-85402,0
C00773=22405,61245,-94532,73319,-125084,-85397,0
C00774=22424,61257,-94500,73306,-125104,-85391,0
C00775=22444,61270,-94466,73292,-125126,-85384,0
C00776=22465,61283,-94432,73278,-125148,-85378,0
C00777=22485,61295,-94397,73264,-125168,-85372,0
C00778=22506,61308,-94363,73250,-125190,-85366,0
C00779=22531,61322,-94324,73232,-125217,-85359,0
C00780=22560,61339,-94280,73211,-125245,-85351,0
C00781=22604,61361,-94221,73178,-125288,-85342,0
C00782=22648,61382,-94162,73145,-125330,-85333,0
C00783=22691,61403,-94107,73113,-125372,-85325,0
C00784=22760,61430,-94032,73058,-125434,-85315,0
C00785=22770,61429,-94036,73048,-125440,-85318,0
C00786=22780,61428,-94039,73037,-125444,-85320,0
C00787=22791,61427,-94043,73026,-125450,-85323,0
C00788=22801,61425,-94047,73015,-125456,-85326,0
C00789=22811,61424,-94050,73004,-125461,-85329,0
C00790=22822,61423,-94054,72993,-125466,-85331,0
C00791=22832,61421,-94057,72982,-125472,-85334,0
C00792=22842,61420,-94061,72971,-125477,-85337,0
C00793=22852,61419,-94065,72961,-125482,-85340,0
C00794=22862,61417,-94070,72950,-125487,-85343,0
C00795=22872,61415,-94074,72940,-125492,-85346,0
C00796=22882,61414,-94079,72929,-125497,-85349,0
C00797=22893,61411,-94085,72917,-125502,-85352,0
C00798=22905,61409,-94093,72903,-125507,-85356,0
C00799=22917,61406,-94100,72890,-125513,-85360,0
C00800=22929,61403,-94107,72876,-125519,-85365,0
C00801=22941,61401,-94115,72863,-125525,-85369,0
C00802=22954,61398,-94122,72850,-125530,-85373,0
C00803=22966,61396,-94129,72836,-125536,-85377,0
C00804=22978,61393,-94137,72823,-125541,-85381,0
C00805=22990,61390,-94144,72809,-125546,-85385,0
C00806=23002,61388,-94151,72796,-125552,-85389,0
C00807=23015,61385,-94159,72782,-125558,-85393,0
C00808=23027,61382,-94166,72769,-125564,-85397,0
C00809=23154,61349,-94258,72626,-125618,-85445,0
C00810=23281,61316,-94350,72482,-125672,-85492,0
C00811=38596,60370,-97191,77203,-121959,-85542,0
C00812=38629,60426,-97035,77194,-122015,-85502,0
C00813=38696,60540,-96721,77179,-122129,-85421,0
C00814=38733,60602,-96552,77170,-122191,-85378,0
C00815=38738,60611,-96528,77169,-122199,-85371,0
C00816=38744,60619,-96504,77167,-122208,-85365,0
C00817=38750,60628,-96480,77165,-122217,-85359,0
C00818=38755,60637,-96456,77163,-122226,-85353,0
C00819=38761,60646,-96432,77162,-122236,-85347,0
C00820=38767,60654,-96407,77160,-122245,-85341,0
C00821=38773,60663,-96384,77158,-122254,-85335,0
C00822=38778,60672,-96359,77157,-122263,-85329,0
C00823=38784,60681,-96335,77155,-122272,-85322,0
C00824=38790,60690,-96311,77153,-122280,-85317,0
C00825=38795,60697,-96291,77151,-122289,-85311,0
C00826=38800,60704,-96271,77149,-122297,-85306,0
C00827=38806,60712,-96250,77147,-122305,-85301,0
C00828=38811,60719,-96230,77145,-122313,-85296,0
C00829=38817,60726,-96210,77143,-122321,-85291,0
C00830=38823,60734,-96191,77141,-122329,-85286,0
C00831=38828,60741,-96171,77138,-122337,-85282,0
C00832=38834,60749,-96148,77136,-122346,-85276,0
C00833=38840,60757,-96125,77135,-122355,-85270,0
C00834=38845,60766,-96102,77132,-122363,-85264,0
C00835=38851,60774,-96079,77131,-122372,-85259,0
C00836=38857,60783,-96056,77129,-122382,-85253,0
C00837=38862,60790,-96035,77127,-122390,-85248,0
C00838=38868,60797,-96016,77125,-122398,-85242,0
C00839=38873,60805,-95996,77122,-122406,-85238,0
C00840=38879,60812,-95977,77120,-122414,-85233,0
C00841=38884,60819,-95957,77118,-122421,-85228,0
C00842=38890,60826,-95938,77116,-122429,-85223,0
C00843=38895,60833,-95918,77114,-122437,-85219,0
C00844=38901,60840,-95900,77111,-122445,-85214,0
C00845=38906,60846,-95882,77109,-122453,-85209,0
C00846=38912,60853,-95863,77106,-122460,-85205,0
C00847=38918,60860,-95845,77104,-122468,-85201,0
C00848=38923,60866,-95827,77101,-122475,-85196,0
C00849=38929,60873,-95809,77099,-122483,-85192,0
C00850=38932,60876,-95800,77097,-122487,-85190,0
C00851=38945,60883,-95782,77087,-122500,-85187,0
C00852=38973,60896,-95747,77066,-122525,-85180,0
C00853=38997,60907,-95717,77047,-122547,-85175,0
C00854=39018,60916,-95693,77031,-122565,-85172,0
C00855=39038,60925,-95670,77015,-122583,-85167,0
C00856=39058,60932,-95649,76999,-122600,-85165,0
C00857=39076,60939,-95631,76984,-122616,-85162,0
C00858=39094,60946,-95612,76970,-122631,-85159,0
C00859=39112,60953,-95594,76955,-122647,-85156,0
C00860=39131,60959,-95575,76940,-122662,-85154,0
C00861=39149,60966,-95557,76925,-122678,-85151,0
C00862=39166,60972,-95541,76911,-122692,-85149,0
C00863=39182,60977,-95528,76898,-122706,-85147,0
C00864=39197,60982,-95514,76885,-122718,-85145,0
C00865=39213,60987,-95500,76872,-122731,-85144,0
C00866=39229,60993,-95486,76859,-122745,-85143,0
C00867=39242,60997,-95476,76848,-122755,-85141,0
C00868=39252,60999,-95468,76839,-122763,-85141,0
C00869=39258,60997,-95476,76832,-122765,-85144,0
C00870=39271,60991,-95492,76817,-122769,-85150,0
C00871=39283,60985,-95508,76803,-122773,-85156,0
C00872=39295,60980,-95524,76788,-122777,-85163,0
C00873=39307,60974,-95539,76774,-122780,-85169,0
C00874=39319,60968,-95555,76759,-122785,-85175,0
C00875=39331,60963,-95571,76745,-122788,-85181,0
C00876=39344,60957,-95587,76730,-122792,-85188,0
C00877=39356,60951,-95604,76715,-122796,-85195,0
C00878=39369,60944,-95623,76700,-122800,-85202,0
C00879=39382,60937,-95641,76684,-122803,-85209,0
C00880=39395,60931,-95660,76668,-122807,-85216,0
C00881=39408,60924,-95679,76653,-122810,-85223,0
C00882=39421,60916,-95700,76636,-122814,-85231,0
C00883=39436,60908,-95724,76617,-122818,-85241,0
C00884=39451,60899,-95748,76599,-122822,-85250,0
C00885=39466,60890,-95772,76580,-122825,-85259,0
C00886=39481,60882,-95796,76561,-122829,-85268,0
C00887=39496,60873,-95820,76543,-122832,-85277,0
C00888=39511,60864,-95845,76524,-122836,-85286,0
C00889=39527,60855,-95871,76505,-122839,-85296,0
C00890=39543,60844,-95900,76484,-122842,-85307,0
C00891=39559,60834,-95929,76463,-122846,-85317,0
C00892=39577,60822,-95963,76440,-122848,-85329,0
C00893=39596,60808,-96001,76415,-122852,-85343,0
C00894=39616,60794,-96039,76390,-122855,-85357,0
C00895=39635,60780,-96078,76364,-122857,-85371,0
C00896=39655,60767,-96116,76339,-122861,-85385,0
C00897=39677,60750,-96163,76309,-122863,-85402,0
C00898=39703,60730,-96219,76275,-122865,-85422,0
C00899=39739,60699,-96305,76225,-122868,-85451,0
C00900=39775,60668,-96391,76176,-122869,-85481,0
C00901=39809,60637,-96477,76128,-122870,-85511,0
C00902=39858,60587,-96615,76057,-122867,-85557,0
C00903=39858,60583,-96627,76054,-122864,-85561,0
C00904=39860,60574,-96651,76049,-122859,-85568,0
C00905=39862,60565,-96676,76043,-122854,-85575,0
C00906=39863,60556,-96700,76038,-122849,-85583,0
C00907=39865,60548,-96724,76032,-122845,-85590,0
C00908=39866,60539,-96748,76027,-122839,-85597,0
C00909=39868,60531,-96770,76022,-122836,-85604,0
C00910=39869,60523,-96792,76017,-122831,-85610,0
C00911=39871,60515,-96814,76012,-122826,-85617,0
C00912=39872,60506,-96838,76006,-122821,-85624,0
C00913=39873,60497,-96863,76001,-122816,-85631,0
C00914=39874,60488,-96887,75996,-122810,-85638,0
C00915=39875,60480,-96912,75991,-122806,-85645,0
C00916=39876,60470,-96939,75986,-122800,-85653,0
C00917=39877,60459,-96970,75980,-122793,-85662,0
C00918=39877,60448,-97000,75974,-122786,-85671,0
C00919=39878,60437,-97030,75969,-122778,-85680,0
C00920=39878,60426,-97061,75963,-122771,-85689,0
C00921=39879,60415,-97091,75958,-122764,-85697,0
C00922=39880,60404,-97121,75952,-122757,-85706,0
C00923=39880,60393,-97152,75946,-122750,-85715,0
C00924=39881,60382,-97182,75941,-122744,-85723,0
C00925=39882,60371,-97212,75935,-122737,-85733,0
C00926=39882,60360,-97243,75930,-122730,-85741,0
C00927=39883,60349,-97273,75924,-122723,-85750,0
C00928=39883,60234,-97593,75871,-122646,-85842,0
C00929=39883,60119,-97912,75819,-122569,-85933,0
C00930=38170,57772,-104527,76515,-119974,-87614,0
C00931=37277,57858,-104259,77453,-119542,-87422,0
C00932=36284,57332,-105767,78242,-118642,-87746,0
C00933=41040,56947,-106991,73225,-120874,-88718,0
C00934=41855,56310,-108897,72094,-120756,-89384,0
C00935=35266,56829,-107223,79076,-117759,-88061,0
C00936=34225,56348,-108626,79952,-116892,-88369,0
C00937=42698,55699,-110753,70936,-120625,-90039,0
C00938=43568,55114,-112561,69751,-120482,-90685,0
C00939=33157,55890,-109978,80872,-116041,-88668,0
C00940=32065,55454,-111279,81834,-115206,-88961,0
C00941=44468,54554,-114322,68536,-120327,-91320,0
C00942=45398,54019,-116035,67292,-120158,-91944,0
C00943=30948,55040,-112528,82837,-114389,-89245,0
C00944=30120,54752,-113404,83593,-113804,-89447,0
C00945=30129,54696,-113577,83566,-113777,-89501,0
C00946=30113,54597,-113884,83553,-113710,-89596,0
C00947=46073,53505,-117705,66326,-119862,-92519,0
C00948=45968,53187,-118740,66295,-119457,-92804,0
C00949=45979,53002,-119351,66199,-119244,-92983,0
C00950=25614,59842,-98444,69367,-125901,-87042,0
C00951=25500,59602,-99112,69361,-125639,-87208,0
C00952=25209,59238,-100129,69476,-125175,-87441,0
C00953=46134,52516,-120980,65811,-118722,-93476,0
C00954=46174,52440,-121238,65734,-118642,-93557,0
C00955=45315,52039,-122587,66494,-117844,-93845,0
C00956=25509,58450,-102367,68769,-124666,-88117,0
C00957=26024,57635,-104715,67824,-124210,-88859,0
C00958=44260,51584,-124150,67448,-116913,-94187,0
C00959=36516,55276,-111909,55193,-126337,-92707,0
C00960=26559,56851,-107012,66872,-123743,-89589,0
C00961=27115,56097,-109258,65910,-123266,-90306,0
C00962=35446,54815,-113308,56151,-125327,-92858,0
C00963=34348,54376,-114657,57151,-124337,-93006,0
C00964=27692,55372,-111457,64936,-122778,-91011,0
C00965=28293,54675,-113611,63949,-122278,-91705,0
C00966=33221,53958,-115956,58192,-123369,-93151,0
C00967=32114,53577,-117155,59230,-122459,-93287,0
C00968=32029,53608,-117054,59339,-122468,-93247,0
C00969=31346,53764,-116539,60169,-122413,-92997,0
C00970=30619,53850,-116252,61010,-122243,-92802,0
C00971=29877,53858,-116211,61828,-121966,-92673,0
C00972=28918,54007,-115721,62948,-121765,-92389,0
C00973=28918,53947,-115744,62958,-121791,-92370,0
C00974=40134,58243,-103073,74762,-121447,-87431,0
C00975=46784,53649,-117086,65658,-120397,-92414,0
C00976=46647,53508,-117537,65742,-120182,-92524,0
C00977=46493,53233,-118426,65783,-119806,-92758,0
C00978=46442,52954,-119343,65710,-119459,-93016,0
C00979=46500,52680,-120252,65522,-119155,-93286,0
C00980=46670,52421,-121128,65220,-118899,-93562,0
C00981=46706,52390,-121235,65166,-118873,-93598,0
C00982=46791,52284,-121596,65025,-118771,-93714,0
C00983=31477,52968,-118950,59678,-121531,-93647,0
C00984=31255,53070,-118611,59972,-121586,-93520,0
C00985=30788,53215,-118129,60557,-121606,-93316,0
C00986=30278,53313,-117801,61165,-121540,-93147,0
C00987=29742,53360,-117640,61776,-121398,-93021,0
C00988=29193,53353,-117652,62374,-121181,-92941,0
C00989=29121,53345,-117677,62449,-121143,-92937,0
C00990=28889,53337,-117700,62699,-121044,-92909,0
C00991=24606,59018,-100611,70027,-124721,-87449,0
C00992=24845,59186,-100142,69864,-124993,-87359,0
C00993=25147,59509,-99242,69715,-125427,-87159,0
C00994=25363,59878,-98214,69682,-125851,-86910,0
C00995=25437,60118,-97549,69730,-126088,-86738,0
C00996=25492,60453,-96623,69847,-126389,-86490,0
C00997=29653,54903,-112770,84137,-113705,-89183,0
C00998=37607,58454,-102423,77397,-120179,-86901,0
C00999=37867,58310,-102837,77078,-120230,-87056,0
//INST
///DATE 2025/02/20 16:20
///COMM Generated using RoboDK
///ATTR SC,RW
///GROUP1 RB1
NOP
MOVL C00000 V=30.0 PL=1
MOVL C00001 V=30.0 PL=1
MOVL C00002 V=30.0 PL=1
MOVL C00003 V=30.0 PL=1
MOVL C00004 V=30.0 PL=1
MOVL C00005 V=30.0 PL=1
MOVL C00006 V=30.0 PL=1
MOVL C00007 V=30.0 PL=1
MOVL C00008 V=30.0 PL=1
MOVL C00009 V=30.0 PL=1
MOVL C00010 V=30.0 PL=1
MOVL C00011 V=30.0 PL=1
MOVL C00012 V=30.0 PL=1
MOVL C00013 V=30.0 PL=1
MOVL C00014 V=30.0 PL=1
MOVL C00015 V=30.0 PL=1
MOVL C00016 V=30.0 PL=1
MOVL C00017 V=30.0 PL=1
MOVL C00018 V=30.0 PL=1
MOVL C00019 V=30.0 PL=1
MOVL C00020 V=30.0 PL=1
MOVL C00021 V=30.0 PL=1
MOVL C00022 V=30.0 PL=1
MOVL C00023 V=30.0 PL=1
MOVL C00024 V=30.0 PL=1
MOVL C00025 V=30.0 PL=1
MOVL C00026 V=30.0 PL=1
MOVL C00027 V=30.0 PL=1
MOVL C00028 V=30.0 PL=1
MOVL C00029 V=30.0 PL=1
MOVL C00030 V=30.0 PL=1
MOVL C00031 V=30.0 PL=1
MOVL C00032 V=30.0 PL=1
MOVL C00033 V=30.0 PL=1
MOVL C00034 V=30.0 PL=1
MOVL C00035 V=30.0 PL=1
MOVL C00036 V=30.0 PL=1
MOVL C00037 V=30.0 PL=1
MOVL C00038 V=30.0 PL=1
MOVL C00039 V=30.0 PL=1
MOVL C00040 V=30.0 PL=1
MOVL C00041 V=30.0 PL=1
MOVL C00042 V=30.0 PL=1
MOVL C00043 V=30.0 PL=1
MOVL C00044 V=30.0 PL=1
MOVL C00045 V=30.0 PL=1
MOVL C00046 V=30.0 PL=1
MOVL C00047 V=30.0 PL=1
MOVL C00048 V=30.0 PL=1
MOVL C00049 V=30.0 PL=1
MOVL C00050 V=30.0 PL=1
MOVL C00051 V=30.0 PL=1
MOVL C00052 V=30.0 PL=1
MOVL C00053 V=30.0 PL=1
MOVL C00054 V=30.0 PL=1
MOVL C00055 V=30.0 PL=1
MOVL C00056 V=30.0 PL=1
MOVL C00057 V=30.0 PL=1
MOVL C00058 V=30.0 PL=1
MOVL C00059 V=30.0 PL=1
MOVL C00060 V=30.0 PL=1
MOVL C00061 V=30.0 PL=1
MOVL C00062 V=30.0 PL=1
MOVL C00063 V=30.0 PL=1
MOVL C00064 V=30.0 PL=1
MOVL C00065 V=30.0 PL=1
MOVL C00066 V=30.0 PL=1
MOVL C00067 V=30.0 PL=1
MOVL C00068 V=30.0 PL=1
MOVL C00069 V=30.0 PL=1
MOVL C00070 V=30.0 PL=1
MOVL C00071 V=30.0 PL=1
MOVL C00072 V=30.0 PL=1
MOVL C00073 V=30.0 PL=1
MOVL C00074 V=30.0 PL=1
MOVL C00075 V=30.0 PL=1
MOVL C00076 V=30.0 PL=1
MOVL C00077 V=30.0 PL=1
MOVL C00078 V=30.0 PL=1
MOVL C00079 V=30.0 PL=1
MOVL C00080 V=30.0 PL=1
MOVL C00081 V=30.0 PL=1
MOVL C00082 V=30.0 PL=1
MOVL C00083 V=30.0 PL=1
MOVL C00084 V=30.0 PL=1
MOVL C00085 V=30.0 PL=1
MOVL C00086 V=30.0 PL=1
MOVL C00087 V=30.0 PL=1
MOVL C00088 V=30.0 PL=1
MOVL C00089 V=30.0 PL=1
MOVL C00090 V=30.0 PL=1
MOVL C00091 V=30.0 PL=1
MOVL C00092 V=30.0 PL=1
MOVL C00093 V=30.0 PL=1
MOVL C00094 V=30.0 PL=1
MOVL C00095 V=30.0 PL=1
MOVL C00096 V=30.0 PL=1
MOVL C00097 V=30.0 PL=1
MOVL C00098 V=30.0 PL=1
MOVL C00099 V=30.0 PL=1
MOVL C00100 V=130.0 PL=1
MOVL C00101 V=30.0 PL=1
MOVL C00102 V=30.0 PL=1
MOVL C00103 V=30.0 PL=1
MOVL C00104 V=30.0 PL=1
MOVL C00105 V=30.0 PL=1
MOVL C00106 V=30.0 PL=1
MOVL C00107 V=30.0 PL=1
MOVL C00108 V=30.0 PL=1
MOVL C00109 V=30.0 PL=1
MOVL C00110 V=30.0 PL=1
MOVL C00111 V=30.0 PL=1
MOVL C00112 V=30.0 PL=1
MOVL C00113 V=30.0 PL=1
MOVL C00114 V=30.0 PL=1
MOVL C00115 V=30.0 PL=1
MOVL C00116 V=30.0 PL=1
MOVL C00117 V=30.0 PL=1
MOVL C00118 V=30.0 PL=1
MOVL C00119 V=30.0 PL=1
MOVL C00120 V=30.0 PL=1
MOVL C00121 V=30.0 PL=1
MOVL C00122 V=30.0 PL=1
MOVL C00123 V=30.0 PL=1
MOVL C00124 V=30.0 PL=1
MOVL C00125 V=30.0 PL=1
MOVL C00126 V=30.0 PL=1
MOVL C00127 V=30.0 PL=1
MOVL C00128 V=30.0 PL=1
MOVL C00129 V=30.0 PL=1
MOVL C00130 V=30.0 PL=1
MOVL C00131 V=30.0 PL=1
MOVL C00132 V=30.0 PL=1
MOVL C00133 V=30.0 PL=1
MOVL C00134 V=30.0 PL=1
MOVL C00135 V=30.0 PL=1
MOVL C00136 V=30.0 PL=1
MOVL C00137 V=30.0 PL=1
MOVL C00138 V=30.0 PL=1
MOVL C00139 V=30.0 PL=1
MOVL C00140 V=30.0 PL=1
MOVL C00141 V=30.0 PL=1
MOVL C00142 V=30.0 PL=1
MOVL C00143 V=30.0 PL=1
MOVL C00144 V=30.0 PL=1
MOVL C00145 V=30.0 PL=1
MOVL C00146 V=30.0 PL=1
MOVL C00147 V=30.0 PL=1
MOVL C00148 V=30.0 PL=1
MOVL C00149 V=30.0 PL=1
MOVL C00150 V=30.0 PL=1
MOVL C00151 V=30.0 PL=1
MOVL C00152 V=30.0 PL=1
MOVL C00153 V=30.0 PL=1
MOVL C00154 V=30.0 PL=1
MOVL C00155 V=30.0 PL=1
MOVL C00156 V=30.0 PL=1
MOVL C00157 V=30.0 PL=1
MOVL C00158 V=30.0 PL=1
MOVL C00159 V=30.0 PL=1
MOVL C00160 V=30.0 PL=1
MOVL C00161 V=30.0 PL=1
MOVL C00162 V=30.0 PL=1
MOVL C00163 V=30.0 PL=1
MOVL C00164 V=30.0 PL=1
MOVL C00165 V=30.0 PL=1
MOVL C00166 V=30.0 PL=1
MOVL C00167 V=30.0 PL=1
MOVL C00168 V=30.0 PL=1
MOVL C00169 V=30.0 PL=1
MOVL C00170 V=30.0 PL=1
MOVL C00171 V=30.0 PL=1
MOVL C00172 V=30.0 PL=1
MOVL C00173 V=30.0 PL=1
MOVL C00174 V=30.0 PL=1
MOVL C00175 V=30.0 PL=1
MOVL C00176 V=30.0 PL=1
MOVL C00177 V=30.0 PL=1
MOVL C00178 V=30.0 PL=1
MOVL C00179 V=30.0 PL=1
MOVL C00180 V=30.0 PL=1
MOVL C00181 V=30.0 PL=1
MOVL C00182 V=30.0 PL=1
MOVL C00183 V=30.0 PL=1
MOVL C00184 V=30.0 PL=1
MOVL C00185 V=30.0 PL=1
MOVL C00186 V=30.0 PL=1
MOVL C00187 V=30.0 PL=1
MOVL C00188 V=30.0 PL=1
MOVL C00189 V=30.0 PL=1
MOVL C00190 V=130.0 PL=1
MOVL C00191 V=30.0 PL=1
MOVL C00192 V=30.0 PL=1
MOVL C00193 V=30.0 PL=1
MOVL C00194 V=30.0 PL=1
MOVL C00195 V=30.0 PL=1
MOVL C00196 V=30.0 PL=1
MOVL C00197 V=30.0 PL=1
MOVL C00198 V=30.0 PL=1
MOVL C00199 V=30.0 PL=1
MOVL C00200 V=30.0 PL=1
MOVL C00201 V=30.0 PL=1
MOVL C00202 V=30.0 PL=1
MOVL C00203 V=30.0 PL=1
MOVL C00204 V=30.0 PL=1
MOVL C00205 V=30.0 PL=1
MOVL C00206 V=30.0 PL=1
MOVL C00207 V=30.0 PL=1
MOVL C00208 V=30.0 PL=1
MOVL C00209 V=30.0 PL=1
MOVL C00210 V=30.0 PL=1
MOVL C00211 V=30.0 PL=1
MOVL C00212 V=30.0 PL=1
MOVL C00213 V=30.0 PL=1
MOVL C00214 V=30.0 PL=1
MOVL C00215 V=30.0 PL=1
MOVL C00216 V=30.0 PL=1
MOVL C00217 V=30.0 PL=1
MOVL C00218 V=30.0 PL=1
MOVL C00219 V=30.0 PL=1
MOVL C00220 V=30.0 PL=1
MOVL C00221 V=30.0 PL=1
MOVL C00222 V=30.0 PL=1
MOVL C00223 V=30.0 PL=1
MOVL C00224 V=30.0 PL=1
MOVL C00225 V=30.0 PL=1
MOVL C00226 V=30.0 PL=1
MOVL C00227 V=30.0 PL=1
MOVL C00228 V=30.0 PL=1
MOVL C00229 V=30.0 PL=1
MOVL C00230 V=30.0 PL=1
MOVL C00231 V=30.0 PL=1
MOVL C00232 V=30.0 PL=1
MOVL C00233 V=30.0 PL=1
MOVL C00234 V=30.0 PL=1
MOVL C00235 V=30.0 PL=1
MOVL C00236 V=30.0 PL=1
MOVL C00237 V=30.0 PL=1
MOVL C00238 V=30.0 PL=1
MOVL C00239 V=30.0 PL=1
MOVL C00240 V=30.0 PL=1
MOVL C00241 V=30.0 PL=1
MOVL C00242 V=30.0 PL=1
MOVL C00243 V=30.0 PL=1
MOVL C00244 V=30.0 PL=1
MOVL C00245 V=30.0 PL=1
MOVL C00246 V=30.0 PL=1
MOVL C00247 V=30.0 PL=1
MOVL C00248 V=30.0 PL=1
MOVL C00249 V=30.0 PL=1
MOVL C00250 V=30.0 PL=1
MOVL C00251 V=30.0 PL=1
MOVL C00252 V=30.0 PL=1
MOVL C00253 V=30.0 PL=1
MOVL C00254 V=30.0 PL=1
MOVL C00255 V=30.0 PL=1
MOVL C00256 V=30.0 PL=1
MOVL C00257 V=30.0 PL=1
MOVL C00258 V=30.0 PL=1
MOVL C00259 V=30.0 PL=1
MOVL C00260 V=30.0 PL=1
MOVL C00261 V=30.0 PL=1
MOVL C00262 V=30.0 PL=1
MOVL C00263 V=30.0 PL=1
MOVL C00264 V=30.0 PL=1
MOVL C00265 V=30.0 PL=1
MOVL C00266 V=30.0 PL=1
MOVL C00267 V=30.0 PL=1
MOVL C00268 V=30.0 PL=1
MOVL C00269 V=30.0 PL=1
MOVL C00270 V=30.0 PL=1
MOVL C00271 V=30.0 PL=1
MOVL C00272 V=30.0 PL=1
MOVL C00273 V=30.0 PL=1
MOVL C00274 V=30.0 PL=1
MOVL C00275 V=30.0 PL=1
MOVL C00276 V=30.0 PL=1
MOVL C00277 V=30.0 PL=1
MOVL C00278 V=30.0 PL=1
MOVL C00279 V=30.0 PL=1
MOVL C00280 V=130.0 PL=1
MOVL C00281 V=20.0 PL=1
MOVL C00282 V=20.0 PL=1
MOVL C00283 V=20.0 PL=1
MOVL C00284 V=20.0 PL=1
MOVL C00285 V=20.0 PL=1
MOVL C00286 V=130.0 PL=1
MOVL C00287 V=20.0 PL=1
MOVL C00288 V=20.0 PL=1
MOVL C00289 V=20.0 PL=1
MOVL C00290 V=20.0 PL=1
MOVL C00291 V=20.0 PL=1
MOVL C00292 V=20.0 PL=1
MOVL C00293 V=20.0 PL=1
MOVL C00294 V=20.0 PL=1
MOVL C00295 V=20.0 PL=1
MOVL C00296 V=20.0 PL=1
MOVL C00297 V=20.0 PL=1
MOVL C00298 V=20.0 PL=1
MOVL C00299 V=20.0 PL=1
MOVL C00300 V=20.0 PL=1
MOVL C00301 V=20.0 PL=1
MOVL C00302 V=20.0 PL=1
MOVL C00303 V=20.0 PL=1
MOVL C00304 V=20.0 PL=1
MOVL C00305 V=20.0 PL=1
MOVL C00306 V=20.0 PL=1
MOVL C00307 V=20.0 PL=1
MOVL C00308 V=20.0 PL=1
MOVL C00309 V=20.0 PL=1
MOVL C00310 V=20.0 PL=1
MOVL C00311 V=20.0 PL=1
MOVL C00312 V=20.0 PL=1
MOVL C00313 V=20.0 PL=1
MOVL C00314 V=20.0 PL=1
MOVL C00315 V=20.0 PL=1
MOVL C00316 V=20.0 PL=1
MOVL C00317 V=20.0 PL=1
MOVL C00318 V=20.0 PL=1
MOVL C00319 V=20.0 PL=1
MOVL C00320 V=20.0 PL=1
MOVL C00321 V=20.0 PL=1
MOVL C00322 V=20.0 PL=1
MOVL C00323 V=130.0 PL=1
MOVL C00324 V=20.0 PL=1
MOVL C00325 V=130.0 PL=1
MOVL C00326 V=130.0 PL=1
MOVL C00327 V=60.0 PL=1
MOVL C00328 V=60.0 PL=1
MOVL C00329 V=60.0 PL=1
MOVL C00330 V=60.0 PL=1
MOVL C00331 V=60.0 PL=1
MOVL C00332 V=60.0 PL=1
MOVL C00333 V=60.0 PL=1
MOVL C00334 V=60.0 PL=1
MOVL C00335 V=60.0 PL=1
MOVL C00336 V=60.0 PL=1
MOVL C00337 V=60.0 PL=1
MOVL C00338 V=60.0 PL=1
MOVL C00339 V=60.0 PL=1
MOVL C00340 V=60.0 PL=1
MOVL C00341 V=60.0 PL=1
MOVL C00342 V=60.0 PL=1
MOVL C00343 V=60.0 PL=1
MOVL C00344 V=60.0 PL=1
MOVL C00345 V=60.0 PL=1
MOVL C00346 V=60.0 PL=1
MOVL C00347 V=60.0 PL=1
MOVL C00348 V=60.0 PL=1
MOVL C00349 V=60.0 PL=1
MOVL C00350 V=60.0 PL=1
MOVL C00351 V=130.0 PL=1
MOVL C00352 V=60.0 PL=1
MOVL C00353 V=60.0 PL=1
MOVL C00354 V=60.0 PL=1
MOVL C00355 V=60.0 PL=1
MOVL C00356 V=60.0 PL=1
MOVL C00357 V=60.0 PL=1
MOVL C00358 V=60.0 PL=1
MOVL C00359 V=60.0 PL=1
MOVL C00360 V=60.0 PL=1
MOVL C00361 V=60.0 PL=1
MOVL C00362 V=60.0 PL=1
MOVL C00363 V=60.0 PL=1
MOVL C00364 V=60.0 PL=1
MOVL C00365 V=60.0 PL=1
MOVL C00366 V=60.0 PL=1
MOVL C00367 V=60.0 PL=1
MOVL C00368 V=60.0 PL=1
MOVL C00369 V=60.0 PL=1
MOVL C00370 V=60.0 PL=1
MOVL C00371 V=60.0 PL=1
MOVL C00372 V=60.0 PL=1
MOVL C00373 V=60.0 PL=1
MOVL C00374 V=60.0 PL=1
MOVL C00375 V=60.0 PL=1
MOVL C00376 V=60.0 PL=1
MOVL C00377 V=60.0 PL=1
MOVL C00378 V=60.0 PL=1
MOVL C00379 V=60.0 PL=1
MOVL C00380 V=60.0 PL=1
MOVL C00381 V=60.0 PL=1
MOVL C00382 V=60.0 PL=1
MOVL C00383 V=60.0 PL=1
MOVL C00384 V=60.0 PL=1
MOVL C00385 V=60.0 PL=1
MOVL C00386 V=60.0 PL=1
MOVL C00387 V=60.0 PL=1
MOVL C00388 V=60.0 PL=1
MOVL C00389 V=60.0 PL=1
MOVL C00390 V=60.0 PL=1
MOVL C00391 V=60.0 PL=1
MOVL C00392 V=60.0 PL=1
MOVL C00393 V=60.0 PL=1
MOVL C00394 V=130.0 PL=1
MOVL C00395 V=30.0 PL=1
MOVL C00396 V=30.0 PL=1
MOVL C00397 V=30.0 PL=1
MOVL C00398 V=30.0 PL=1
MOVL C00399 V=30.0 PL=1
MOVL C00400 V=30.0 PL=1
MOVL C00401 V=30.0 PL=1
MOVL C00402 V=30.0 PL=1
MOVL C00403 V=30.0 PL=1
MOVL C00404 V=30.0 PL=1
MOVL C00405 V=30.0 PL=1
MOVL C00406 V=30.0 PL=1
MOVL C00407 V=30.0 PL=1
MOVL C00408 V=30.0 PL=1
MOVL C00409 V=30.0 PL=1
MOVL C00410 V=30.0 PL=1
MOVL C00411 V=30.0 PL=1
MOVL C00412 V=30.0 PL=1
MOVL C00413 V=30.0 PL=1
MOVL C00414 V=30.0 PL=1
MOVL C00415 V=30.0 PL=1
MOVL C00416 V=30.0 PL=1
MOVL C00417 V=30.0 PL=1
MOVL C00418 V=30.0 PL=1
MOVL C00419 V=30.0 PL=1
MOVL C00420 V=30.0 PL=1
MOVL C00421 V=30.0 PL=1
MOVL C00422 V=30.0 PL=1
MOVL C00423 V=30.0 PL=1
MOVL C00424 V=30.0 PL=1
MOVL C00425 V=30.0 PL=1
MOVL C00426 V=30.0 PL=1
MOVL C00427 V=30.0 PL=1
MOVL C00428 V=30.0 PL=1
MOVL C00429 V=30.0 PL=1
MOVL C00430 V=30.0 PL=1
MOVL C00431 V=30.0 PL=1
MOVL C00432 V=30.0 PL=1
MOVL C00433 V=30.0 PL=1
MOVL C00434 V=30.0 PL=1
MOVL C00435 V=30.0 PL=1
MOVL C00436 V=30.0 PL=1
MOVL C00437 V=30.0 PL=1
MOVL C00438 V=30.0 PL=1
MOVL C00439 V=30.0 PL=1
MOVL C00440 V=30.0 PL=1
MOVL C00441 V=30.0 PL=1
MOVL C00442 V=30.0 PL=1
MOVL C00443 V=30.0 PL=1
MOVL C00444 V=30.0 PL=1
MOVL C00445 V=30.0 PL=1
MOVL C00446 V=30.0 PL=1
MOVL C00447 V=30.0 PL=1
MOVL C00448 V=30.0 PL=1
MOVL C00449 V=30.0 PL=1
MOVL C00450 V=30.0 PL=1
MOVL C00451 V=30.0 PL=1
MOVL C00452 V=30.0 PL=1
MOVL C00453 V=30.0 PL=1
MOVL C00454 V=30.0 PL=1
MOVL C00455 V=30.0 PL=1
MOVL C00456 V=30.0 PL=1
MOVL C00457 V=30.0 PL=1
MOVL C00458 V=30.0 PL=1
MOVL C00459 V=30.0 PL=1
MOVL C00460 V=30.0 PL=1
MOVL C00461 V=30.0 PL=1
MOVL C00462 V=30.0 PL=1
MOVL C00463 V=30.0 PL=1
MOVL C00464 V=30.0 PL=1
MOVL C00465 V=30.0 PL=1
MOVL C00466 V=30.0 PL=1
MOVL C00467 V=130.0 PL=1
MOVL C00468 V=130.0 PL=1
MOVL C00469 V=30.0 PL=1
MOVL C00470 V=30.0 PL=1
MOVL C00471 V=30.0 PL=1
MOVL C00472 V=30.0 PL=1
MOVL C00473 V=30.0 PL=1
MOVL C00474 V=30.0 PL=1
MOVL C00475 V=30.0 PL=1
MOVL C00476 V=30.0 PL=1
MOVL C00477 V=30.0 PL=1
MOVL C00478 V=30.0 PL=1
MOVL C00479 V=30.0 PL=1
MOVL C00480 V=30.0 PL=1
MOVL C00481 V=30.0 PL=1
MOVL C00482 V=30.0 PL=1
MOVL C00483 V=30.0 PL=1
MOVL C00484 V=30.0 PL=1
MOVL C00485 V=30.0 PL=1
MOVL C00486 V=30.0 PL=1
MOVL C00487 V=30.0 PL=1
MOVL C00488 V=30.0 PL=1
MOVL C00489 V=30.0 PL=1
MOVL C00490 V=30.0 PL=1
MOVL C00491 V=30.0 PL=1
MOVL C00492 V=30.0 PL=1
MOVL C00493 V=30.0 PL=1
MOVL C00494 V=30.0 PL=1
MOVL C00495 V=30.0 PL=1
MOVL C00496 V=30.0 PL=1
MOVL C00497 V=30.0 PL=1
MOVL C00498 V=30.0 PL=1
MOVL C00499 V=30.0 PL=1
MOVL C00500 V=30.0 PL=1
MOVL C00501 V=30.0 PL=1
MOVL C00502 V=30.0 PL=1
MOVL C00503 V=30.0 PL=1
MOVL C00504 V=30.0 PL=1
MOVL C00505 V=30.0 PL=1
MOVL C00506 V=30.0 PL=1
MOVL C00507 V=30.0 PL=1
MOVL C00508 V=30.0 PL=1
MOVL C00509 V=30.0 PL=1
MOVL C00510 V=30.0 PL=1
MOVL C00511 V=30.0 PL=1
MOVL C00512 V=30.0 PL=1
MOVL C00513 V=30.0 PL=1
MOVL C00514 V=30.0 PL=1
MOVL C00515 V=30.0 PL=1
MOVL C00516 V=30.0 PL=1
MOVL C00517 V=30.0 PL=1
MOVL C00518 V=30.0 PL=1
MOVL C00519 V=30.0 PL=1
MOVL C00520 V=30.0 PL=1
MOVL C00521 V=30.0 PL=1
MOVL C00522 V=30.0 PL=1
MOVL C00523 V=30.0 PL=1
MOVL C00524 V=30.0 PL=1
MOVL C00525 V=30.0 PL=1
MOVL C00526 V=30.0 PL=1
MOVL C00527 V=30.0 PL=1
MOVL C00528 V=30.0 PL=1
MOVL C00529 V=30.0 PL=1
MOVL C00530 V=30.0 PL=1
MOVL C00531 V=30.0 PL=1
MOVL C00532 V=30.0 PL=1
MOVL C00533 V=30.0 PL=1
MOVL C00534 V=30.0 PL=1
MOVL C00535 V=30.0 PL=1
MOVL C00536 V=30.0 PL=1
MOVL C00537 V=30.0 PL=1
MOVL C00538 V=30.0 PL=1
MOVL C00539 V=30.0 PL=1
MOVL C00540 V=30.0 PL=1
MOVL C00541 V=30.0 PL=1
MOVL C00542 V=30.0 PL=1
MOVL C00543 V=30.0 PL=1
MOVL C00544 V=30.0 PL=1
MOVL C00545 V=30.0 PL=1
MOVL C00546 V=30.0 PL=1
MOVL C00547 V=30.0 PL=1
MOVL C00548 V=30.0 PL=1
MOVL C00549 V=30.0 PL=1
MOVL C00550 V=30.0 PL=1
MOVL C00551 V=30.0 PL=1
MOVL C00552 V=30.0 PL=1
MOVL C00553 V=30.0 PL=1
MOVL C00554 V=30.0 PL=1
MOVL C00555 V=30.0 PL=1
MOVL C00556 V=30.0 PL=1
MOVL C00557 V=30.0 PL=1
MOVL C00558 V=30.0 PL=1
MOVL C00559 V=30.0 PL=1
MOVL C00560 V=30.0 PL=1
MOVL C00561 V=30.0 PL=1
MOVL C00562 V=30.0 PL=1
MOVL C00563 V=30.0 PL=1
MOVL C00564 V=30.0 PL=1
MOVL C00565 V=30.0 PL=1
MOVL C00566 V=30.0 PL=1
MOVL C00567 V=30.0 PL=1
MOVL C00568 V=30.0 PL=1
MOVL C00569 V=30.0 PL=1
MOVL C00570 V=30.0 PL=1
MOVL C00571 V=30.0 PL=1
MOVL C00572 V=30.0 PL=1
MOVL C00573 V=30.0 PL=1
MOVL C00574 V=30.0 PL=1
MOVL C00575 V=30.0 PL=1
MOVL C00576 V=30.0 PL=1
MOVL C00577 V=30.0 PL=1
MOVL C00578 V=30.0 PL=1
MOVL C00579 V=30.0 PL=1
MOVL C00580 V=130.0 PL=1
MOVL C00581 V=30.0 PL=1
MOVL C00582 V=30.0 PL=1
MOVL C00583 V=30.0 PL=1
MOVL C00584 V=30.0 PL=1
MOVL C00585 V=30.0 PL=1
MOVL C00586 V=30.0 PL=1
MOVL C00587 V=30.0 PL=1
MOVL C00588 V=30.0 PL=1
MOVL C00589 V=30.0 PL=1
MOVL C00590 V=30.0 PL=1
MOVL C00591 V=30.0 PL=1
MOVL C00592 V=30.0 PL=1
MOVL C00593 V=30.0 PL=1
MOVL C00594 V=30.0 PL=1
MOVL C00595 V=30.0 PL=1
MOVL C00596 V=30.0 PL=1
MOVL C00597 V=30.0 PL=1
MOVL C00598 V=30.0 PL=1
MOVL C00599 V=30.0 PL=1
MOVL C00600 V=30.0 PL=1
MOVL C00601 V=30.0 PL=1
MOVL C00602 V=30.0 PL=1
MOVL C00603 V=30.0 PL=1
MOVL C00604 V=30.0 PL=1
MOVL C00605 V=30.0 PL=1
MOVL C00606 V=30.0 PL=1
MOVL C00607 V=30.0 PL=1
MOVL C00608 V=30.0 PL=1
MOVL C00609 V=30.0 PL=1
MOVL C00610 V=30.0 PL=1
MOVL C00611 V=30.0 PL=1
MOVL C00612 V=30.0 PL=1
MOVL C00613 V=30.0 PL=1
MOVL C00614 V=30.0 PL=1
MOVL C00615 V=30.0 PL=1
MOVL C00616 V=30.0 PL=1
MOVL C00617 V=30.0 PL=1
MOVL C00618 V=30.0 PL=1
MOVL C00619 V=30.0 PL=1
MOVL C00620 V=30.0 PL=1
MOVL C00621 V=30.0 PL=1
MOVL C00622 V=30.0 PL=1
MOVL C00623 V=30.0 PL=1
MOVL C00624 V=30.0 PL=1
MOVL C00625 V=30.0 PL=1
MOVL C00626 V=30.0 PL=1
MOVL C00627 V=30.0 PL=1
MOVL C00628 V=30.0 PL=1
MOVL C00629 V=30.0 PL=1
MOVL C00630 V=30.0 PL=1
MOVL C00631 V=30.0 PL=1
MOVL C00632 V=30.0 PL=1
MOVL C00633 V=30.0 PL=1
MOVL C00634 V=30.0 PL=1
MOVL C00635 V=30.0 PL=1
MOVL C00636 V=30.0 PL=1
MOVL C00637 V=30.0 PL=1
MOVL C00638 V=30.0 PL=1
MOVL C00639 V=30.0 PL=1
MOVL C00640 V=30.0 PL=1
MOVL C00641 V=30.0 PL=1
MOVL C00642 V=30.0 PL=1
MOVL C00643 V=30.0 PL=1
MOVL C00644 V=30.0 PL=1
MOVL C00645 V=30.0 PL=1
MOVL C00646 V=30.0 PL=1
MOVL C00647 V=30.0 PL=1
MOVL C00648 V=30.0 PL=1
MOVL C00649 V=30.0 PL=1
MOVL C00650 V=30.0 PL=1
MOVL C00651 V=30.0 PL=1
MOVL C00652 V=30.0 PL=1
MOVL C00653 V=30.0 PL=1
MOVL C00654 V=30.0 PL=1
MOVL C00655 V=30.0 PL=1
MOVL C00656 V=30.0 PL=1
MOVL C00657 V=30.0 PL=1
MOVL C00658 V=30.0 PL=1
MOVL C00659 V=30.0 PL=1
MOVL C00660 V=30.0 PL=1
MOVL C00661 V=30.0 PL=1
MOVL C00662 V=30.0 PL=1
MOVL C00663 V=30.0 PL=1
MOVL C00664 V=30.0 PL=1
MOVL C00665 V=30.0 PL=1
MOVL C00666 V=30.0 PL=1
MOVL C00667 V=30.0 PL=1
MOVL C00668 V=30.0 PL=1
MOVL C00669 V=30.0 PL=1
MOVL C00670 V=30.0 PL=1
MOVL C00671 V=30.0 PL=1
MOVL C00672 V=30.0 PL=1
MOVL C00673 V=30.0 PL=1
MOVL C00674 V=30.0 PL=1
MOVL C00675 V=30.0 PL=1
MOVL C00676 V=30.0 PL=1
MOVL C00677 V=30.0 PL=1
MOVL C00678 V=30.0 PL=1
MOVL C00679 V=30.0 PL=1
MOVL C00680 V=30.0 PL=1
MOVL C00681 V=30.0 PL=1
MOVL C00682 V=30.0 PL=1
MOVL C00683 V=30.0 PL=1
MOVL C00684 V=30.0 PL=1
MOVL C00685 V=30.0 PL=1
MOVL C00686 V=30.0 PL=1
MOVL C00687 V=30.0 PL=1
MOVL C00688 V=30.0 PL=1
MOVL C00689 V=30.0 PL=1
MOVL C00690 V=30.0 PL=1
MOVL C00691 V=30.0 PL=1
MOVL C00692 V=30.0 PL=1
MOVL C00693 V=130.0 PL=1
MOVL C00694 V=30.0 PL=1
MOVL C00695 V=30.0 PL=1
MOVL C00696 V=30.0 PL=1
MOVL C00697 V=30.0 PL=1
MOVL C00698 V=30.0 PL=1
MOVL C00699 V=30.0 PL=1
MOVL C00700 V=30.0 PL=1
MOVL C00701 V=30.0 PL=1
MOVL C00702 V=30.0 PL=1
MOVL C00703 V=30.0 PL=1
MOVL C00704 V=30.0 PL=1
MOVL C00705 V=30.0 PL=1
MOVL C00706 V=30.0 PL=1
MOVL C00707 V=30.0 PL=1
MOVL C00708 V=30.0 PL=1
MOVL C00709 V=30.0 PL=1
MOVL C00710 V=30.0 PL=1
MOVL C00711 V=30.0 PL=1
MOVL C00712 V=30.0 PL=1
MOVL C00713 V=30.0 PL=1
MOVL C00714 V=30.0 PL=1
MOVL C00715 V=30.0 PL=1
MOVL C00716 V=30.0 PL=1
MOVL C00717 V=30.0 PL=1
MOVL C00718 V=30.0 PL=1
MOVL C00719 V=30.0 PL=1
MOVL C00720 V=30.0 PL=1
MOVL C00721 V=30.0 PL=1
MOVL C00722 V=30.0 PL=1
MOVL C00723 V=30.0 PL=1
MOVL C00724 V=30.0 PL=1
MOVL C00725 V=30.0 PL=1
MOVL C00726 V=30.0 PL=1
MOVL C00727 V=30.0 PL=1
MOVL C00728 V=30.0 PL=1
MOVL C00729 V=30.0 PL=1
MOVL C00730 V=30.0 PL=1
MOVL C00731 V=30.0 PL=1
MOVL C00732 V=30.0 PL=1
MOVL C00733 V=30.0 PL=1
MOVL C00734 V=30.0 PL=1
MOVL C00735 V=30.0 PL=1
MOVL C00736 V=30.0 PL=1
MOVL C00737 V=30.0 PL=1
MOVL C00738 V=30.0 PL=1
MOVL C00739 V=30.0 PL=1
MOVL C00740 V=30.0 PL=1
MOVL C00741 V=30.0 PL=1
MOVL C00742 V=30.0 PL=1
MOVL C00743 V=30.0 PL=1
MOVL C00744 V=30.0 PL=1
MOVL C00745 V=30.0 PL=1
MOVL C00746 V=30.0 PL=1
MOVL C00747 V=30.0 PL=1
MOVL C00748 V=30.0 PL=1
MOVL C00749 V=30.0 PL=1
MOVL C00750 V=30.0 PL=1
MOVL C00751 V=30.0 PL=1
MOVL C00752 V=30.0 PL=1
MOVL C00753 V=30.0 PL=1
MOVL C00754 V=30.0 PL=1
MOVL C00755 V=30.0 PL=1
MOVL C00756 V=30.0 PL=1
MOVL C00757 V=30.0 PL=1
MOVL C00758 V=30.0 PL=1
MOVL C00759 V=30.0 PL=1
MOVL C00760 V=30.0 PL=1
MOVL C00761 V=30.0 PL=1
MOVL C00762 V=30.0 PL=1
MOVL C00763 V=30.0 PL=1
MOVL C00764 V=30.0 PL=1
MOVL C00765 V=30.0 PL=1
MOVL C00766 V=30.0 PL=1
MOVL C00767 V=30.0 PL=1
MOVL C00768 V=30.0 PL=1
MOVL C00769 V=30.0 PL=1
MOVL C00770 V=30.0 PL=1
MOVL C00771 V=30.0 PL=1
MOVL C00772 V=30.0 PL=1
MOVL C00773 V=30.0 PL=1
MOVL C00774 V=30.0 PL=1
MOVL C00775 V=30.0 PL=1
MOVL C00776 V=30.0 PL=1
MOVL C00777 V=30.0 PL=1
MOVL C00778 V=30.0 PL=1
MOVL C00779 V=30.0 PL=1
MOVL C00780 V=30.0 PL=1
MOVL C00781 V=30.0 PL=1
MOVL C00782 V=30.0 PL=1
MOVL C00783 V=30.0 PL=1
MOVL C00784 V=30.0 PL=1
MOVL C00785 V=30.0 PL=1
MOVL C00786 V=30.0 PL=1
MOVL C00787 V=30.0 PL=1
MOVL C00788 V=30.0 PL=1
MOVL C00789 V=30.0 PL=1
MOVL C00790 V=30.0 PL=1
MOVL C00791 V=30.0 PL=1
MOVL C00792 V=30.0 PL=1
MOVL C00793 V=30.0 PL=1
MOVL C00794 V=30.0 PL=1
MOVL C00795 V=30.0 PL=1
MOVL C00796 V=30.0 PL=1
MOVL C00797 V=30.0 PL=1
MOVL C00798 V=30.0 PL=1
MOVL C00799 V=30.0 PL=1
MOVL C00800 V=30.0 PL=1
MOVL C00801 V=30.0 PL=1
MOVL C00802 V=30.0 PL=1
MOVL C00803 V=30.0 PL=1
MOVL C00804 V=30.0 PL=1
MOVL C00805 V=30.0 PL=1
MOVL C00806 V=30.0 PL=1
MOVL C00807 V=30.0 PL=1
MOVL C00808 V=30.0 PL=1
MOVL C00809 V=30.0 PL=1
MOVL C00810 V=30.0 PL=1
MOVL C00811 V=130.0 PL=1
MOVL C00812 V=30.0 PL=1
MOVL C00813 V=30.0 PL=1
MOVL C00814 V=30.0 PL=1
MOVL C00815 V=30.0 PL=1
MOVL C00816 V=30.0 PL=1
MOVL C00817 V=30.0 PL=1
MOVL C00818 V=30.0 PL=1
MOVL C00819 V=30.0 PL=1
MOVL C00820 V=30.0 PL=1
MOVL C00821 V=30.0 PL=1
MOVL C00822 V=30.0 PL=1
MOVL C00823 V=30.0 PL=1
MOVL C00824 V=30.0 PL=1
MOVL C00825 V=30.0 PL=1
MOVL C00826 V=30.0 PL=1
MOVL C00827 V=30.0 PL=1
MOVL C00828 V=30.0 PL=1
MOVL C00829 V=30.0 PL=1
MOVL C00830 V=30.0 PL=1
MOVL C00831 V=30.0 PL=1
MOVL C00832 V=30.0 PL=1
MOVL C00833 V=30.0 PL=1
MOVL C00834 V=30.0 PL=1
MOVL C00835 V=30.0 PL=1
MOVL C00836 V=30.0 PL=1
MOVL C00837 V=30.0 PL=1
MOVL C00838 V=30.0 PL=1
MOVL C00839 V=30.0 PL=1
MOVL C00840 V=30.0 PL=1
MOVL C00841 V=30.0 PL=1
MOVL C00842 V=30.0 PL=1
MOVL C00843 V=30.0 PL=1
MOVL C00844 V=30.0 PL=1
MOVL C00845 V=30.0 PL=1
MOVL C00846 V=30.0 PL=1
MOVL C00847 V=30.0 PL=1
MOVL C00848 V=30.0 PL=1
MOVL C00849 V=30.0 PL=1
MOVL C00850 V=30.0 PL=1
MOVL C00851 V=30.0 PL=1
MOVL C00852 V=30.0 PL=1
MOVL C00853 V=30.0 PL=1
MOVL C00854 V=30.0 PL=1
MOVL C00855 V=30.0 PL=1
MOVL C00856 V=30.0 PL=1
MOVL C00857 V=30.0 PL=1
MOVL C00858 V=30.0 PL=1
MOVL C00859 V=30.0 PL=1
MOVL C00860 V=30.0 PL=1
MOVL C00861 V=30.0 PL=1
MOVL C00862 V=30.0 PL=1
MOVL C00863 V=30.0 PL=1
MOVL C00864 V=30.0 PL=1
MOVL C00865 V=30.0 PL=1
MOVL C00866 V=30.0 PL=1
MOVL C00867 V=30.0 PL=1
MOVL C00868 V=30.0 PL=1
MOVL C00869 V=30.0 PL=1
MOVL C00870 V=30.0 PL=1
MOVL C00871 V=30.0 PL=1
MOVL C00872 V=30.0 PL=1
MOVL C00873 V=30.0 PL=1
MOVL C00874 V=30.0 PL=1
MOVL C00875 V=30.0 PL=1
MOVL C00876 V=30.0 PL=1
MOVL C00877 V=30.0 PL=1
MOVL C00878 V=30.0 PL=1
MOVL C00879 V=30.0 PL=1
MOVL C00880 V=30.0 PL=1
MOVL C00881 V=30.0 PL=1
MOVL C00882 V=30.0 PL=1
MOVL C00883 V=30.0 PL=1
MOVL C00884 V=30.0 PL=1
MOVL C00885 V=30.0 PL=1
MOVL C00886 V=30.0 PL=1
MOVL C00887 V=30.0 PL=1
MOVL C00888 V=30.0 PL=1
MOVL C00889 V=30.0 PL=1
MOVL C00890 V=30.0 PL=1
MOVL C00891 V=30.0 PL=1
MOVL C00892 V=30.0 PL=1
MOVL C00893 V=30.0 PL=1
MOVL C00894 V=30.0 PL=1
MOVL C00895 V=30.0 PL=1
MOVL C00896 V=30.0 PL=1
MOVL C00897 V=30.0 PL=1
MOVL C00898 V=30.0 PL=1
MOVL C00899 V=30.0 PL=1
MOVL C00900 V=30.0 PL=1
MOVL C00901 V=30.0 PL=1
MOVL C00902 V=30.0 PL=1
MOVL C00903 V=30.0 PL=1
MOVL C00904 V=30.0 PL=1
MOVL C00905 V=30.0 PL=1
MOVL C00906 V=30.0 PL=1
MOVL C00907 V=30.0 PL=1
MOVL C00908 V=30.0 PL=1
MOVL C00909 V=30.0 PL=1
MOVL C00910 V=30.0 PL=1
MOVL C00911 V=30.0 PL=1
MOVL C00912 V=30.0 PL=1
MOVL C00913 V=30.0 PL=1
MOVL C00914 V=30.0 PL=1
MOVL C00915 V=30.0 PL=1
MOVL C00916 V=30.0 PL=1
MOVL C00917 V=30.0 PL=1
MOVL C00918 V=30.0 PL=1
MOVL C00919 V=30.0 PL=1
MOVL C00920 V=30.0 PL=1
MOVL C00921 V=30.0 PL=1
MOVL C00922 V=30.0 PL=1
MOVL C00923 V=30.0 PL=1
MOVL C00924 V=30.0 PL=1
MOVL C00925 V=30.0 PL=1
MOVL C00926 V=30.0 PL=1
MOVL C00927 V=30.0 PL=1
MOVL C00928 V=30.0 PL=1
MOVL C00929 V=30.0 PL=1
MOVL C00930 V=130.0 PL=1
MOVL C00931 V=20.0 PL=1
MOVL C00932 V=20.0 PL=1
MOVL C00933 V=20.0 PL=1
MOVL C00934 V=20.0 PL=1
MOVL C00935 V=20.0 PL=1
MOVL C00936 V=20.0 PL=1
MOVL C00937 V=20.0 PL=1
MOVL C00938 V=20.0 PL=1
MOVL C00939 V=20.0 PL=1
MOVL C00940 V=20.0 PL=1
MOVL C00941 V=20.0 PL=1
MOVL C00942 V=20.0 PL=1
MOVL C00943 V=20.0 PL=1
MOVL C00944 V=20.0 PL=1
MOVL C00945 V=20.0 PL=1
MOVL C00946 V=20.0 PL=1
MOVL C00947 V=20.0 PL=1
MOVL C00948 V=20.0 PL=1
MOVL C00949 V=20.0 PL=1
MOVL C00950 V=20.0 PL=1
MOVL C00951 V=20.0 PL=1
MOVL C00952 V=20.0 PL=1
MOVL C00953 V=20.0 PL=1
MOVL C00954 V=20.0 PL=1
MOVL C00955 V=20.0 PL=1
MOVL C00956 V=20.0 PL=1
MOVL C00957 V=20.0 PL=1
MOVL C00958 V=20.0 PL=1
MOVL C00959 V=20.0 PL=1
MOVL C00960 V=20.0 PL=1
MOVL C00961 V=20.0 PL=1
MOVL C00962 V=20.0 PL=1
MOVL C00963 V=20.0 PL=1
MOVL C00964 V=20.0 PL=1
MOVL C00965 V=20.0 PL=1
MOVL C00966 V=20.0 PL=1
MOVL C00967 V=20.0 PL=1
MOVL C00968 V=20.0 PL=1
MOVL C00969 V=20.0 PL=1
MOVL C00970 V=20.0 PL=1
MOVL C00971 V=20.0 PL=1
MOVL C00972 V=20.0 PL=1
MOVL C00973 V=130.0 PL=1
MOVL C00974 V=130.0 PL=1
MOVL C00975 V=60.0 PL=1
MOVL C00976 V=60.0 PL=1
MOVL C00977 V=60.0 PL=1
MOVL C00978 V=60.0 PL=1
MOVL C00979 V=60.0 PL=1
MOVL C00980 V=60.0 PL=1
MOVL C00981 V=60.0 PL=1
MOVL C00982 V=60.0 PL=1
MOVL C00983 V=60.0 PL=1
MOVL C00984 V=60.0 PL=1
MOVL C00985 V=60.0 PL=1
MOVL C00986 V=60.0 PL=1
MOVL C00987 V=60.0 PL=1
MOVL C00988 V=60.0 PL=1
MOVL C00989 V=60.0 PL=1
MOVL C00990 V=60.0 PL=1
MOVL C00991 V=60.0 PL=1
MOVL C00992 V=60.0 PL=1
MOVL C00993 V=60.0 PL=1
MOVL C00994 V=60.0 PL=1
MOVL C00995 V=60.0 PL=1
MOVL C00996 V=60.0 PL=1
MOVL C00997 V=60.0 PL=1
MOVL C00998 V=60.0 PL=1
MOVL C00999 V=60.0 PL=1
END
